	ChannelType												: UDINT := 1;(*  NC channel type:
																								1	Stantard,
																								2	Interpreter (CNC)
																								3	FIFO 
																								4	Kinematic *) 
                                        					
	EncType													: 	UDINT := E_NcEncoderType.NcEncoderType_undefined;(* Encoder type: - See property with E_NcEncoderType data type *)																																									
	EncTypAbs												:	BOOL := 0; (* Encodertyp Abs = 1/ Rel = 0*)
	
	DriveType												:	UDINT := TO_UDINT(E_NcDriveType.NcDriveType_undefined);
	
	RefFlag													:	BOOL := 0; (* Axis is in reference *)
                                							
	LimitPosActive											: 	BOOL;
	LimitNegActive											:	BOOL;
	LimitPos												: 	LREAL;
	LimitNeg												: 	LREAL;

	TargetPosWindow											:	LREAL;
	TargetPosWindowMonitoring								:	BOOL;
	PosRangeWindow											: 	LREAL;
	PosRangeWindowMonitoring								:	BOOL;
                                							
	DynamicsRefVelocity										: 	LREAL;
	DynamicsMaxVelocity										: 	LREAL;
	G0Velocity												: 	LREAL;
	RefVelocityPos											: 	LREAL;
	RefVelocityNeg											: 	LREAL;
	ManVelocityFast											: 	LREAL;
	ManVelocitySlow											: 	LREAL;
                                							  	
	Kv														: 	LREAL;
	Jerk													: 	LREAL;
	Acc														: 	LREAL;
	Dec														: 	LREAL;
	MaxPosLagValue											: 	LREAL;
	MaxPosLagFilterTime										: 	LREAL;
	MaxPosLagMonitoring										: 	BOOL;
                                                              	
	InvertEncCoutingDir										: 	BOOL;
	ModuloFactor											: 	LREAL;
	ToleranceWindowModuloStart								: 	LREAL;
	EncScalingNumerator										:	LREAL;
	EncScalingDenominator									:	LREAL;
	EncScaling												: 	LREAL; //Factor of Numerator and Denominator
	PosBias													: 	LREAL;  (* Actual NC position offset *)
	ReferenceSystem											:	UDINT; //incremental, absolute
	CalibrationMode											:	UDINT;
	CalibrationValue										: 	LREAL;	(* read/write only allowed for certain encoder types  *)
	RefFlagDistance											: 	LREAL;	(* read/write only allowed for certain encoder types *)
	CalibrInvertDirForCamSearch								:	BOOL; (* TRUE=Cam search direction negative , read/write only allowed for certain encoder types *)
	CalibrInvertDirForSyncImpSearch							:	BOOL; (* TRUE=Sync impuls (off cam) search direction negative, read/write only allowed for certain encoder types *)

	InvertMotorPolarity										: 	BOOL;
                                							  	
	BreakingDistancePos										: 	LREAL;
	BreakingDistanceNeg										: 	LREAL;
	
	PhysicalUnit											:	STRING[10+1];
END_VAR                         	


VAR
(* Zwischenspeicher ************************************************************)
	
(* Deklaration Trigger **********************************************************)

(* Zeiten ******************************************************************)

(* Bausteine ***************************************************************)
	ReadAdsPara												: ADSREAD := (NetId	:= '' , Port := AMSPORT_R0_NC, TmOut	:= DEFAULT_ADS_TIMEOUT);
	WriteAdsPara											: ADSWRITE := (NetId:= '' , Port := AMSPORT_R0_NC, TmOut	:= DEFAULT_ADS_TIMEOUT);

(* Dummy Speicher **********************************************************)

END_VAR

	(************************************************************************************)
	(*																					*)
	(*		B E C K H O F F   N E W   A U T O M A T I O N   T E C H N O L O G Y    		*)
	(*																					*)
	(*		Eiserstr.5	D-33415 Verl	Germany	phone:	+49-5246-0	www.Beckhoff.Com	*)
    (*																					*)
    (*		Bausteinbeschreibung	:	Read/Write axis parameter						*)
	(*		TwinCAT-Version			:	3.x or higher									*)
	(*																					*)
	(************************************************************************************)

(* Execute ***************************************************************************************)
	Super^();			
	
(*************************************************************************************************)

PROPERTY PROTECTED deviceAddrIsValid : BOOL
GET
deviceAddrIsValid := AxisId > 0;
END_GET
END_PROPERTY

PROPERTY PUBLIC eAxisType : E_NcAxisType
GET
eAxisType := AxisType;
END_GET
END_PROPERTY

PROPERTY PUBLIC eDriveType : E_NcDriveType
GET
eDriveType := DriveType;
END_GET
END_PROPERTY

PROPERTY PUBLIC eEncType : E_NcEncoderType
GET
eEncType := EncType;
END_GET
END_PROPERTY

METHOD PROTECTED getValue : BOOL //Return value = TRUE if execution finished and state incremented 
VAR_INPUT
	IDxGrp						:	UDINT;
	IDxOffs						:	UDINT;
	Len							:	UDINT;
	pActValue					:	PVOID; //Address of variable for actual value
	pSetValue					:	PVOID; //Address of variable for ser value variable, can be zero if no corresponding SetVariable exists
END_VAR

ReadAdsPara	(Read := TRUE, IDxGrp:=IDxGrp+AxisId, IDxOffs:=IDxOffs,LEN:=Len,DestAddr:=pActValue );
IF NOT ReadAdsPara.BUSY
THEN
	IF NOT ReadAdsPara.ERR 
	THEN 
		IF pSetValue <> 0 THEN MEMCPY(pSetValue, pActValue, Len); END_IF			
		state 												:= state + 1; 
	ELSE 		
		Busy												:= FALSE;
		Error												:= TRUE;
		ErrorId												:= ReadAdsPara.ERRID;
		ErrorText											:= CONCAT('Error read parameter in state:' , TO_STRING(state * -1));
		ErrorText											:= CONCAT(ErrorText , ' Id:');
		ErrorText											:= CONCAT(ErrorText , TO_STRING(ErrorId));
		State												:= 9999;
	END_IF	
	ReadAdsPara(Read := FALSE); 
	getValue												:= TRUE;									
END_IF
END_METHOD

METHOD PROTECTED seqRead : BOOL //Return value = TRUE if execution finished 
VAR_IN_OUT
	State							:	INT;
END_VAR
(* Execute read axis parameter ************************************)
	CASE state OF
	1..99: //read application spec parameter 
		seqRead												:= TRUE;
		
	1001: (* Name *************************************************************************************)
		IF LEN(Name) > 0 AND NOT ReadAdsPara.BUSY
		THEN
			state											:= state + 1;
		ELSE
			getValue(IDxGrp:= 16#4000,	IDxOffs := 16#2,	LEN := SIZEOF(Name),		pActValue := ADR(Name),			pSetValue := 0);
		END_IF

	1002: (* Axis Type ( Für Beschreibung Typen siehe AxPara) **********************************)
		IF AxisType <> 0 AND NOT ReadAdsPara.BUSY
		THEN
			state											:= state + 1;
		ELSE
			getValue(IDxGrp:= 16#4000,	IDxOffs := 16#3,	LEN := SIZEOF(AxisType),	pActValue := ADR(AxisType), 	pSetValue := 0);
		END_IF

	1003: (* NC Channel type ****************************************************************************************)
		IF ChannelType <> 0 AND NOT ReadAdsPara.BUSY
		THEN
			state											:= state + 1;
		ELSE
			getValue(IDxGrp:= 16#4000,	IDxOffs := 16#53,	LEN := SIZEOF(ChannelType),	pActValue := ADR(ChannelType), 	pSetValue := 0);
		END_IF

	1004: (* EncType ****************************************************************************************)
		IF EncType <> 0 AND NOT ReadAdsPara.BUSY
		THEN
			state											:= state + 1;
		ELSE
			getValue(IDxGrp:= 16#5000,	IDxOffs := 16#3,	LEN := SIZEOF(EncType),	pActValue := ADR(EncType), 		pSetValue := 0);
		END_IF
	
	1005: (* Endlagenlimit pos. ***********************************************************************)
		getValue(IDxGrp:= 16#5000,	IDxOffs := 16#E,	LEN := SIZEOF(LimitPos),	pActValue := ADR(LimitPos),  pSetValue := ADR(SetLimitPos) );	
	
	1006: (* Endlagenlimit neg ***********************************************************************)
		getValue(IDxGrp:= 16#5000,	IDxOffs := 16#D,	LEN := SIZEOF(LimitNeg),	pActValue := ADR(LimitNeg),  pSetValue := ADR(SetLimitNeg) );
		
	1007: (* Endlagenlimit pos aktiv ? ***************************************************************)
		IF getValue(IDxGrp:= 16#5000,	IDxOffs := 16#C,	LEN := SIZEOF(_UINT),	pActValue := ADR(_UINT),  pSetValue := 0)
		THEN
			SetLimitPosActive :=LimitPosActive				:= TO_BOOL(_UINT);
		END_IF

	1008: (* Endlagenlimit neg aktiv ? ***************************************************************)
		IF getValue(IDxGrp:= 16#5000,	IDxOffs := 16#B,	LEN := SIZEOF(_UINT),	pActValue := ADR(_UINT),  pSetValue := 0)
		THEN
			SetLimitNegActive :=LimitNegActive				:= TO_BOOL(_UINT);
		END_IF

	1009: (* Zielfenster ******************************************************************************)
		getValue(IDxGrp:= 16#4000,	IDxOffs := 16#16,	LEN := SIZEOF(TargetPosWindow),	pActValue := ADR(TargetPosWindow),  pSetValue := ADR(SetTargetPosWindow) );

	1010: (* Positionsfenster ************************************************************************)
		getValue(IDxGrp:= 16#4000,	IDxOffs := 16#10,	LEN := SIZEOF(PosRangeWindow),	pActValue := ADR(PosRangeWindow),  pSetValue := ADR(SetPosRangeWindow) );

	1011: (* Bezugsgeschwindigkeit (siehe Typenschild)*************************************)
		IF AxisType = 2 
		THEN
			state											:= state + 1;
		ELSE
			getValue(IDxGrp:= 16#7000,	IDxOffs := 16#101,	LEN := SIZEOF(DynamicsRefVelocity),	pActValue := ADR(DynamicsRefVelocity),  pSetValue := ADR(SetDynamicsRefVelocity) );
		END_IF
	
	1012: (* Max.Geschwindigkeit (ca. 90% der Bezugsgeschw.)***************************)
		IF AxisType = 2 
		THEN
			state											:= state + 1;
		ELSE
			getValue(IDxGrp:= 16#4000,	IDxOffs := 16#27,	LEN := SIZEOF(DynamicsMaxVelocity),	pActValue := ADR(DynamicsMaxVelocity),  pSetValue := ADR(SetDynamicsMaxVelocity) );
		END_IF
		
	1013: (* G0 Geschwindigkeit ****************************************************************)
		getValue(IDxGrp:= 16#4000,	IDxOffs := 16#A,	LEN := SIZEOF(G0Velocity),	pActValue := ADR(G0Velocity),  pSetValue := ADR(SetG0Velocity) );

	1014: (* Ref.Geschwindigkeit Pos **********************************************************)
		getValue(IDxGrp:= 16#4000,	IDxOffs := 16#6,	LEN := SIZEOF(RefVelocityPos),	pActValue := ADR(RefVelocityPos),  pSetValue := ADR(SetRefVelocityPos) );

	1015: (* Ref.Geschwindigkeit Neg **********************************************************)
		getValue(IDxGrp:= 16#4000,	IDxOffs := 16#7,	LEN := SIZEOF(RefVelocityNeg),	pActValue := ADR(RefVelocityNeg),  pSetValue := ADR(SetRefVelocityNeg) );

	1016: (* Man. Verfahrgeschwindigkeit fast *************************************************)
		getValue(IDxGrp:= 16#4000,	IDxOffs := 16#9,	LEN := SIZEOF(ManVelocityFast),	pActValue := ADR(ManVelocityFast),  pSetValue := ADR(SetManVelocityFast) );

	1017: (* Man. Verfahrgeschwindigkeit slow ***********************************************)
		getValue(IDxGrp:= 16#4000,	IDxOffs := 16#8,	LEN := SIZEOF(ManVelocitySlow),	pActValue := ADR(ManVelocitySlow),  pSetValue := ADR(SetManVelocitySlow) );

	1018: (* Kv ************************************************************************************)
		IF AxisType = 2
		THEN
			state											:= state + 1;
		ELSE
			getValue(IDxGrp:= 16#6000,	IDxOffs := 16#102,	LEN := SIZEOF(Kv),	pActValue := ADR(Kv),  pSetValue := ADR(SetKv) );
		END_IF

	1019: (* Ruck ************************************************************************************)
		IF AxisType = 2 
		THEN
			state											:= state + 1;
		ELSE
			getValue(IDxGrp:= 16#4000,	IDxOffs := 16#103,	LEN := SIZEOF(Jerk),	pActValue := ADR(Jerk),  pSetValue := ADR(SetJerk) );
		END_IF
		

	1020: (* Beschleunigung ***********************************************************************)
		IF AxisType = 2
		THEN
			state											:= state + 1;
		ELSE
			getValue(IDxGrp:= 16#4000,	IDxOffs := 16#101,	LEN := SIZEOF(Acc),	pActValue := ADR(Acc),  pSetValue := ADR(SetAcc) );
		END_IF

	1021: (* Verzoegerung ***************************************************************************)
		IF AxisType = 2 
		then
			state											:= state + 1;
		ELSE
			getValue(IDxGrp:= 16#4000,	IDxOffs := 16#102,	LEN := SIZEOF(Dec),	pActValue := ADR(Dec),  pSetValue := ADR(SetDec) );
		END_IF

	1022: (* Schleppabstand ***********************************************************************)	
		getValue(IDxGrp:= 16#6000,	IDxOffs := 16#12,	LEN := SIZEOF(MaxPosLagValue),	pActValue := ADR(MaxPosLagValue),  pSetValue := ADR(SetMaxPosLagValue) );

	1023: (* Skalierung ******************************************************************************)
		getValue(IDxGrp:= 16#5000,	IDxOffs := 16#6,	LEN := SIZEOF(EncScaling),	pActValue := ADR(EncScaling),  pSetValue := 0 );		

	1024: (* Positions Offset  ***********************************************************************)
		getValue(IDxGrp:= 16#5000,	IDxOffs := 16#7,	LEN := SIZEOF(PosBias),	pActValue := ADR(PosBias),  pSetValue := ADR(SetPosBias) );

	1025: (* Referenzposition (Nicht bei Absolut Encoder lesen)*******************************)
		IF EncType <> 2 AND EncType <> 5 AND EncType<> 7 AND EncType <> 11 AND EncType <> 12
		THEN
			getValue(IDxGrp:= 16#5000,	IDxOffs := 16#103,	LEN := SIZEOF(CalibrationValue),	pActValue := ADR(CalibrationValue),  pSetValue := ADR(SetCalibrationValue) );
		ELSE
			state											:= state +1;
		END_IF

	1026: (* Abstand Ref-Nocken Synchronimpuls (Nicht bei Absolut Encoder lesen) ****)
		IF EncType <> 2 AND EncType <> 5 AND EncType <> 7 AND EncType <> 11 AND EncType <> 12
		THEN
			getValue(IDxGrp:= 16#5100,	IDxOffs := 16#101,	LEN := SIZEOF(RefFlagDistance),	pActValue := ADR(RefFlagDistance),  pSetValue := 0 );
		ELSE
			state											:= state +1;
		END_IF

	1027: (* Drive direction **************************************************************)
		IF getValue(IDxGrp:= 16#7000,	IDxOffs := 16#6,	LEN := SIZEOF(_UINT),	pActValue := ADR(_UINT),  pSetValue := 0)
		THEN
			SetInvertMotorPolarity :=InvertMotorPolarity	:= TO_BOOL(_UINT);
			
		END_IF

	1028: (* Bremsweg positiv **********************************************************************)
		IF AxisType <> 2
		THEN
			state											:= state + 1;
		ELSE
			getValue(IDxGrp:= 16#4000,	IDxOffs := 16#303,	LEN := SIZEOF(BreakingDistancePos),	pActValue := ADR(BreakingDistancePos),  pSetValue := ADR(SetBreakingDistancePos ));
		END_IF

	1029: (* Bremsweg negativ *********************************************************************)
		IF AxisType <> 2 
		THEN
			state											:= state + 1;
		ELSE
			getValue(IDxGrp:= 16#4000,	IDxOffs := 16#304,	LEN := SIZEOF(BreakingDistanceNeg),	pActValue := ADR(BreakingDistanceNeg),  pSetValue := ADR(SetBreakingDistanceNeg ));

		END_IF

	1030: (* Schleppueberwachung Aktiv *********************************************************************)
		IF getValue(IDxGrp:= 16#6000,	IDxOffs := 16#10,	LEN := SIZEOF(_UINT),	pActValue := ADR(_UINT),  pSetValue := 0)
		THEN
			SetMaxPosLagMonitoring :=MaxPosLagMonitoring	:= TO_BOOL(_UINT);
			
		END_IF

	1031: (* Encodertyp Abs/Rel *********************************************************************)
		IF getValue(IDxGrp:= 16#5000,	IDxOffs := 16#1D,	LEN := SIZEOF(_UINT),	pActValue := ADR(_UINT),  pSetValue := 0)
		THEN
			EncTypAbs										:= TO_BOOL(_UINT);
			
		END_IF

	1032: (* Referenzierflag *********************************************************************)
		IF getValue(IDxGrp:= 16#5100,	IDxOffs := 16#9,	LEN := SIZEOF(_UINT),	pActValue := ADR(_UINT),  pSetValue := 0)
		THEN
			SetRefFlag :=RefFlag							:= TO_BOOL(_UINT);
		END_IF

	1033: (* Zielfenster Aktiv ******************************************************************)
		IF getValue(IDxGrp:= 16#4000,	IDxOffs := 16#15,	LEN := SIZEOF(_UINT),	pActValue := ADR(_UINT),  pSetValue := 0)
		THEN
			SetTargetPosWindowMonitoring :=TargetPosWindowMonitoring := TO_BOOL(_UINT);
			
		END_IF

	1034: (* Positionsfenster Aktiv ******************************************************************)
		IF getValue(IDxGrp:= 16#4000,	IDxOffs := 16#F,	LEN := SIZEOF(_UINT),	pActValue := ADR(_UINT),  pSetValue := 0)
		THEN
			SetPosRangeWindowMonitoring :=PosRangeWindowMonitoring := TO_BOOL(_UINT);
			
		END_IF

	1035: (* ModuloFaktor ******************************************************************)
		getValue(IDxGrp:= 16#5000,	IDxOffs := 16#9,	LEN := SIZEOF(ModuloFactor),	pActValue := ADR(ModuloFactor),  pSetValue := ADR(SetModuloFactor ));

	1036: (* Enc Zaehlrichtung ******************************************************************)
		IF getValue(IDxGrp:= 16#5000,	IDxOffs := 16#8,	LEN := SIZEOF(_UINT),	pActValue := ADR(_UINT),  pSetValue := 0)
		THEN
			SetInvertEncCoutingDir :=InvertEncCoutingDir := TO_BOOL(_UINT);
			
		END_IF

	1037: (* Toleranzfenster Modulo Start *******************************************************)
		getValue(IDxGrp:= 16#5000,	IDxOffs := 16#1B,	LEN := SIZEOF(ToleranceWindowModuloStart),	pActValue := ADR(ToleranceWindowModuloStart),  pSetValue := ADR(SetToleranceWindowModuloStart ));
		
	1038: (* Calibration cam search direction inverted *******************************************************)
		IF EncType <> 2 AND EncType <> 5 AND EncType<> 7 AND EncType <> 11 AND EncType <> 12
		THEN
			IF getValue(IDxGrp:= 16#5000,	IDxOffs := 16#101,	LEN := SIZEOF(_UINT),	pActValue := ADR(_UINT),  pSetValue := 0)
			THEN
				SetCalibrInvertDirForCamSearch :=CalibrInvertDirForCamSearch := TO_BOOL(_UINT);
				
			END_IF
		ELSE
			state											:= state +1;
		END_IF		
		
	1039: (* Calibration impuls direction inverted (of cam) *******************************************************)
		IF EncType <> 2 AND EncType <> 5 AND EncType<> 7 AND EncType <> 11 AND EncType <> 12
		THEN
			IF getValue(IDxGrp:= 16#5000,	IDxOffs := 16#102,	LEN := SIZEOF(_UINT),	pActValue := ADR(_UINT),  pSetValue := 0)
			THEN
				SetCalibrInvertDirForSyncImpSearch :=CalibrInvertDirForSyncImpSearch := TO_BOOL(_UINT);
				
			END_IF
	
		ELSE
			state											:= state +1;
		END_IF	
		
	1040: (* Calibration mode *******************************************************)
		IF EncType <> 2 AND EncType <> 5 AND EncType<> 7 AND EncType <> 11 AND EncType <> 12
		THEN
			getValue(IDxGrp:= 16#5000,	IDxOffs := 16#107,	LEN := SIZEOF(CalibrationMode),	pActValue := ADR(CalibrationMode),  pSetValue := ADR(SetCalibrationMode));
		ELSE
			state											:= state +1;
		END_IF
		
	1041: (* Scaling numerator **************************************)
		getValue(IDxGrp:= 16#5000,	IDxOffs := 16#23,	LEN := SIZEOF(EncScalingNumerator),	pActValue := ADR(EncScalingNumerator),  pSetValue := ADR(SetEncScalingNumerator) );	
			
	1042: (* Scaling denumerator **************************************)
		getValue(IDxGrp:= 16#5000,	IDxOffs := 16#24,	LEN := SIZEOF(EncScalingDenominator),	pActValue := ADR(EncScalingDenominator),  pSetValue := ADR(SetEncScalingDenominator) );	
		
	1043: (* Reference system **************************************)
		getValue(IDxGrp:= 16#5000,	IDxOffs := 16#19,	LEN := SIZEOF(ReferenceSystem),	pActValue := ADR(ReferenceSystem),  pSetValue := ADR(SetReferenceSystem) );	

	1044: (* Schleppabstand Filter Time ***********************************************************************)	
		getValue(IDxGrp:= 16#6000,	IDxOffs := 16#13,	LEN := SIZEOF(MaxPosLagFilterTime),	pActValue := ADR(MaxPosLagFilterTime),  pSetValue := ADR(SetMaxPosLagFilterTime) );

	1045: (* Physical unit ***********************************************************************)	
		getValue(IDxGrp:= 16#4000,	IDxOffs := 16#5,	LEN := SIZEOF(PhysicalUnit),	pActValue := ADR(PhysicalUnit),  pSetValue := ADR(PhysicalUnit) );
		IF PhysicalUnit[0] = 176 THEN PhysicalUnit := '°'; END_IF		
		
	1046: (*  Drive type ***********************************************************************)	
		getValue(IDxGrp:= 16#7000,	IDxOffs := 16#3,	LEN := SIZEOF(DriveType),	pActValue := ADR(DriveType),  pSetValue := 0 );
			
	ELSE
		state												:= 1;
	END_CASE

(*********************************************************************************************)
END_METHOD

METHOD PROTECTED seqWrite : BOOL //Return value = TRUE if execution finished 
VAR_IN_OUT
	State							:	INT;
END_VAR
(* Write axis parameter ********************************************************************)
	CASE state OF
	1..99: //Wite application spec parameter 
		seqWrite											:= TRUE;
		
	1001: (* Endlagenlimit pos.beschreiben ********************************************************)
		setValue(IDxGrp:= 16#5000,	IDxOffs := 16#E,	LEN := SIZEOF(SetLimitPos),		pActValue := ADR(LimitPos),		pSetValue := ADR(SetLimitPos));

	1002: (* Endlagenlimit neg.beschreiben ********************************************************)
		setValue(IDxGrp:= 16#5000,	IDxOffs := 16#D,	LEN := SIZEOF(SetLimitNeg),		pActValue := ADR(LimitNeg),		pSetValue := ADR(SetLimitNeg));

	1003: (* Endlagenlimit pos. aktiv ****************************************************************)
		IF NOT (SetLimitPosActive XOR LimitPosActive)
			AND NOT WriteAdsPara.BUSY
		THEN 
			state 											:= state + 1;
		ELSE
			_UINT											:= TO_UINT(SetLimitPosActive);
			LimitPosActive									:= SetLimitPosActive;
			setValue(IDxGrp:= 16#5000,	IDxOffs := 16#C,	LEN := SIZEOF(_UINT),		pActValue := 0,		pSetValue := ADR(_UINT));
		END_IF
		
	1004: (* Endlagenlimit neg.aktiv *****************************************************************)
		IF NOT (SetLimitNegActive XOR LimitNegActive) 
			AND NOT WriteAdsPara.BUSY
		THEN 
			state 											:= state + 1;
		ELSE
			_UINT											:= TO_UINT(SetLimitNegActive);
			LimitNegActive									:= SetLimitNegActive; 
			setValue(IDxGrp:= 16#5000,	IDxOffs := 16#B,	LEN := SIZEOF(_UINT),		pActValue := 0,		pSetValue := ADR(_UINT));
		END_IF

	1005: (* Zielfenster setzen **********************************************************************)
		setValue(IDxGrp:= 16#4000,	IDxOffs := 16#16,	LEN := SIZEOF(SetTargetPosWindow),		pActValue := ADR(TargetPosWindow),		pSetValue := ADR(SetTargetPosWindow));

	1006: (* Positionsfenster setzen *****************************************************************)
		setValue(IDxGrp:= 16#4000,	IDxOffs := 16#10,	LEN := SIZEOF(SetPosRangeWindow),		pActValue := ADR(PosRangeWindow),	pSetValue := ADR(SetPosRangeWindow));
		
	1007: (* Bezugsgeschwindigkeit setzen ********************************************************)
		IF AxisType = 2
		THEN 
			state 											:= state +1;
		ELSE
			setValue(IDxGrp:= 16#7000,	IDxOffs := 16#101,	LEN := SIZEOF(SetDynamicsRefVelocity),pActValue := ADR(DynamicsRefVelocity),	pSetValue := ADR(SetDynamicsRefVelocity));
		END_IF


	1008: (* Max.Geschwindigkeit setzen ************************************************************)
		IF AxisType = 2 
		THEN 
			state 											:= state +1;
		ELSE
			setValue(IDxGrp:= 16#4000,	IDxOffs := 16#27,	LEN := SIZEOF(SetDynamicsMaxVelocity),pActValue := ADR(DynamicsMaxVelocity),	pSetValue := ADR(SetDynamicsMaxVelocity));
		END_IF

	1009: (* G0 Geschwindigkeit setzen ****************************************************************)
		setValue(IDxGrp:= 16#4000,	IDxOffs := 16#A,	LEN := SIZEOF(SetG0Velocity),	pActValue := ADR(G0Velocity),	pSetValue := ADR(SetG0Velocity));

	1010: (* Ref.Geschwindigkeit fast setzen *******************************************************)
		setValue(IDxGrp:= 16#4000,	IDxOffs := 16#6,	LEN := SIZEOF(SetRefVelocityPos),	pActValue := ADR(RefVelocityPos),	pSetValue := ADR(SetRefVelocityPos));

	1011: (* Ref.Geschwindigkeit slow setzen *****************************************************)
		setValue(IDxGrp:= 16#4000,	IDxOffs := 16#7,	LEN := SIZEOF(SetRefVelocityNeg),	pActValue := ADR(RefVelocityNeg),	pSetValue := ADR(SetRefVelocityNeg));

	1012: (* Man.Geschwindigkeit fast setzen ******************************************************)
		setValue(IDxGrp:= 16#4000,	IDxOffs := 16#9,	LEN := SIZEOF(SetManVelocityFast),	pActValue := ADR(ManVelocityFast),	pSetValue := ADR(SetManVelocityFast));
		

	1013: (* Man.Geschwindigkeit slow setzen ******************************************************)
		setValue(IDxGrp:= 16#4000,	IDxOffs := 16#8,	LEN := SIZEOF(SetManVelocitySlow),	pActValue := ADR(ManVelocitySlow),	pSetValue := ADR(SetManVelocitySlow));

	1014: (* Kv setzen **************************************************************************************)
		IF AxisType = 2 
		THEN 
			state 											:= state +1;
		ELSE
			setValue(IDxGrp:= 16#6000,	IDxOffs := 16#102,	LEN := SIZEOF(SetKv),pActValue := ADR(Kv),	pSetValue := ADR(SetKv));
		END_IF

	1015: (* Ruck setzen ***********************************************************************************)
		IF AxisType = 2 
		THEN 
			state 											:= state +1;
		ELSE
			setValue(IDxGrp:= 16#4000,	IDxOffs := 16#103,	LEN := SIZEOF(SetJerk),pActValue := ADR(Jerk),	pSetValue := ADR(SetJerk));
		END_IF

	1016: (* Beschleunigung setzen **********************************************************************)
		IF AxisType = 2 
		THEN 
			state 											:= state +1;
		ELSE
			setValue(IDxGrp:= 16#4000,	IDxOffs := 16#101,	LEN := SIZEOF(SetAcc), pActValue := ADR(Acc),	pSetValue := ADR(SetAcc));
		END_IF
	
	1017: (* Verzoegerung setzen ************************************************************************)
		IF AxisType = 2 
		THEN 
			state 											:= state +1;
		ELSE
			setValue(IDxGrp:= 16#4000,	IDxOffs := 16#102,	LEN := SIZEOF(SetDec), pActValue := ADR(Dec),	pSetValue := ADR(SetDec));
		END_IF
		
	1018: (* Schleppabstand setzen **********************************************************************)
		setValue(IDxGrp:= 16#6000,	IDxOffs := 16#12,	LEN := SIZEOF(SetMaxPosLagValue),	pActValue := ADR(MaxPosLagValue),	pSetValue := ADR(SetMaxPosLagValue));

	1019: (* Reserverd *****************************************************************************)
		// Set scaling replaced by Num and Denum  setValue(IDxGrp:= 16#5000,	IDxOffs := 16#6,	LEN := SIZEOF(SetEncScaling),	pActValue := ADR(EncScaling),	pSetValue := ADR(SetEncScaling));
		state 												:= state +1 ;
		
	1020: (* Positions Offset setzen ****************************************************************)
		setValue(IDxGrp:= 16#5000,	IDxOffs := 16#7,	LEN := SIZEOF(SetPosBias),	pActValue := ADR(PosBias),	pSetValue := ADR(SetPosBias));
		
	1021: (* Referenzposition setzen ***************************************************************)
		IF EncType <> 2  AND EncType <> 5 AND EncType <> 7 AND EncType <> 11  AND EncType <> 12 
		THEN
			setValue(IDxGrp:= 16#5000,	IDxOffs := 16#103,	LEN := SIZEOF(SetCalibrationValue),	pActValue := ADR(CalibrationValue),	pSetValue := ADR(SetCalibrationValue));
		ELSE
			state 											:= state +1 ;
		END_IF

	1022: (* Bremsweg positiv **********************************************************************)
		IF AxisType = 2 
		THEN 
			state 											:= state +1;
		ELSE
			setValue(IDxGrp:= 16#4000,	IDxOffs := 16#303,	LEN := SIZEOF(SetBreakingDistancePos), pActValue := ADR(BreakingDistancePos),	pSetValue := ADR(SetBreakingDistancePos));
		END_IF

	1023: (* Bremsweg negativ *********************************************************************)
		IF AxisType = 2
		THEN 
			state 											:= state +1;
		ELSE
			setValue(IDxGrp:= 16#4000,	IDxOffs := 16#304,	LEN := SIZEOF(SetBreakingDistanceNeg), pActValue := ADR(BreakingDistanceNeg),	pSetValue := ADR(SetBreakingDistanceNeg));
		END_IF

	1024: (* Schleppueberwachung ****************************************************************************)
		IF SetMaxPosLagMonitoring = MaxPosLagMonitoring AND NOT WriteAdsPara.BUSY
		THEN 
			state 											:= state +1;
		ELSE
			_UINT											:= TO_UINT(SetMaxPosLagMonitoring);
			MaxPosLagMonitoring								:= SetMaxPosLagMonitoring;					
			setValue(IDxGrp:= 16#6000,	IDxOffs := 16#10,	LEN := SIZEOF(_UINT),	pActValue := 0,	pSetValue := ADR(_UINT));
		END_IF

	1025: (* Referenzierflag ****************************************************************************)
		IF RefFlag = SetRefFlag AND NOT WriteAdsPara.BUSY
		THEN 
			state 											:= state +1;
		ELSE
			_UINT											:= TO_UINT(SetRefFlag);
			RefFlag											:= SetRefFlag;
			setValue(IDxGrp:= 16#5100,	IDxOffs := 16#9,	LEN := SIZEOF(_UINT), pActValue := 0,	pSetValue := ADR(_UINT));
		END_IF
		
	1026: (* PosfensterAktiv ****************************************************************************)
		IF SetPosRangeWindowMonitoring = PosRangeWindowMonitoring AND NOT WriteAdsPara.BUSY
		THEN 
			state 											:= state +1;
		ELSE
			_UINT											:= TO_UINT(SetPosRangeWindowMonitoring);
			PosRangeWindowMonitoring						:= SetPosRangeWindowMonitoring;
			setValue(IDxGrp:= 16#4000,	IDxOffs := 16#F,	LEN := SIZEOF(_UINT), pActValue := 0,	pSetValue := ADR(_UINT));
		END_IF

	1027: (* ZielfensterAktiv ****************************************************************************)
		IF SetTargetPosWindowMonitoring = TargetPosWindowMonitoring AND NOT WriteAdsPara.BUSY
		THEN 
			state 											:= state +1;
		ELSE
			_UINT											:= TO_UINT(SetTargetPosWindowMonitoring);
			TargetPosWindowMonitoring						:= SetTargetPosWindowMonitoring;
			setValue(IDxGrp:= 16#4000,	IDxOffs := 16#15,	LEN := SIZEOF(_UINT), pActValue := 0,	pSetValue := ADR(_UINT));
		END_IF

	1028: (* Modulofaktor ****************************************************************************)
		setValue(IDxGrp:= 16#5000,	IDxOffs := 16#9,	LEN := SIZEOF(SetModuloFactor), pActValue := ADR(ModuloFactor),	pSetValue := ADR(SetModuloFactor));
		
	1029: (* Enc. Zaehlrichtung ****************************************************************************)
		IF SetInvertEncCoutingDir = InvertEncCoutingDir AND NOT WriteAdsPara.BUSY
		THEN 
			state 											:= state +1;
		ELSE
			_UINT											:= TO_UINT(SetInvertEncCoutingDir);
			InvertEncCoutingDir								:= SetInvertEncCoutingDir;
			setValue(IDxGrp:= 16#5000,	IDxOffs := 16#8,	LEN := SIZEOF(_UINT), pActValue := 0,	pSetValue := ADR(_UINT));
		END_IF

	1030: (* Drive  ****************************************************************************)
		IF SetInvertMotorPolarity = InvertMotorPolarity AND NOT WriteAdsPara.BUSY
		THEN 
			state 											:= state +1;
		ELSE
			_UINT											:= TO_UINT(SetInvertMotorPolarity);
			InvertMotorPolarity								:= SetInvertMotorPolarity;
			setValue(IDxGrp:= 16#7000,	IDxOffs := 16#6,	LEN := SIZEOF(_UINT), pActValue := 0,	pSetValue := ADR(_UINT));
		END_IF
		
		
	1031: (* Enc. Modulo start tolerance ****************************************************************************)
		setValue(IDxGrp:= 16#5000,	IDxOffs := 16#1B,	LEN := SIZEOF(SetToleranceWindowModuloStart), pActValue := ADR(ToleranceWindowModuloStart),	pSetValue := ADR(SetToleranceWindowModuloStart));

	1032: (* Set calibration cam search direction inverted ***************************************************************)
		IF SetCalibrInvertDirForCamSearch = CalibrInvertDirForCamSearch	AND NOT WriteAdsPara.BUSY
			OR_ELSE(EncType = 2  OR EncType = 5 OR EncType = 7 OR EncType = 11  OR EncType = 12)
		THEN 
			state 											:= state +1;
		ELSE
			_UINT											:= TO_UINT(SetCalibrInvertDirForCamSearch);
			CalibrInvertDirForCamSearch						:= SetCalibrInvertDirForCamSearch;
			setValue(IDxGrp:= 16#5000,	IDxOffs := 16#101,	LEN := SIZEOF(_UINT), pActValue := 0,	pSetValue := ADR(_UINT));
		END_IF

	1033: (* Set calibration impuls search direction inverted ***************************************************************)
		IF SetCalibrInvertDirForSyncImpSearch = CalibrInvertDirForSyncImpSearch AND NOT WriteAdsPara.BUSY
			OR_ELSE(EncType = 2  OR EncType = 5 OR EncType = 7 OR EncType = 11  OR EncType = 12)
		THEN 
			state 											:= state +1;
		ELSE
			_UINT											:= TO_UINT(SetCalibrInvertDirForSyncImpSearch);
			CalibrInvertDirForSyncImpSearch					:= SetCalibrInvertDirForSyncImpSearch;
			setValue(IDxGrp:= 16#5000,	IDxOffs := 16#102,	LEN := SIZEOF(_UINT), pActValue := 0,	pSetValue := ADR(_UINT));
		END_IF
		
	1034: (* Set calibration mode ***************************************************************)
		IF SetCalibrationMode = CalibrationMode  AND NOT WriteAdsPara.BUSY
			OR_ELSE(EncType = 2  OR EncType = 5 OR EncType = 7 OR EncType = 11  OR EncType = 12)
		THEN 
			state 											:= state +1;		
		ELSE
			setValue(IDxGrp:= 16#5000,	IDxOffs := 16#107,	LEN := SIZEOF(SetCalibrationMode), pActValue := ADR(CalibrationMode),	pSetValue := ADR(SetCalibrationMode));
		END_IF

	1035: (* Scaling numerator **************************************)
		setValue(IDxGrp:= 16#5000,	IDxOffs := 16#23,	LEN := SIZEOF(SetEncScalingNumerator),	pActValue := ADR(EncScalingNumerator),  pSetValue := ADR(SetEncScalingNumerator) );	
			
	1036: (* Scaling denumerator **************************************)
		setValue(IDxGrp:= 16#5000,	IDxOffs := 16#24,	LEN := SIZEOF(SetEncScalingDenominator),	pActValue := ADR(EncScalingDenominator),  pSetValue := ADR(SetEncScalingDenominator) );
		
		//Calculate Act Scaling 
		IF NOT Error THEN  EncScaling	:= EncScalingNumerator / EncScalingDenominator; END_IF
		
	1037: (* Reference system **************************************)
		setValue(IDxGrp:= 16#5000,	IDxOffs := 16#19,	LEN := SIZEOF(SetReferenceSystem),	pActValue := ADR(ReferenceSystem),  pSetValue := ADR(SetReferenceSystem) );	
	
	1038: (* Schleppueberwachung Zeit ****************************************************************************)
		setValue(IDxGrp:= 16#6000,	IDxOffs := 16#13,	LEN := SIZEOF(SetMaxPosLagFilterTime),	pActValue := ADR(MaxPosLagFilterTime),	pSetValue := ADR(SetMaxPosLagFilterTime));
	
	ELSE
		state 												:= 1 ;
	END_CASE
	
(***********************************************************************************************)
END_METHOD

METHOD PROTECTED setValue : BOOL //Return value = TRUE if execution finished and state incremented 
VAR_INPUT
	IDxGrp						:	UDINT;
	IDxOffs						:	UDINT;
	Len							:	UDINT;
	pActValue					:	PVOID; //Address of variable for actual value, can be zero if no corresponding acual value variable exists
	pSetValue					:	PVOID; //Address of variable for set value variable
END_VAR

IF pActValue <> 0 AND pSetValue <> 0 AND_THEN MEMCMP(pSetValue, pActValue, Len) = 0
THEN //Skip write parameter if set and actual value are equel
	state													:= state + 1;	
	setValue												:= TRUE;
ELSE
	WriteAdsPara( Write := TRUE, IdxGrp :=IDxGrp+AxisId, IdxOffs:=IDxOffs, LEN:=Len, SrcAddr:=pSetValue );
	IF NOT WriteAdsPara.BUSY
	THEN
		IF NOT WriteAdsPara.ERR
		THEN
			IF pActValue <> 0 THEN MEMCPY(pActValue, pSetValue, Len); END_IF	
			state											:= state + 1;
		ELSE
			Busy											:= FALSE;
			Error											:= TRUE;
			ErrorId											:= WriteAdsPara.ERRID;
			ErrorText										:= CONCAT('Error write parameter in state:' , TO_STRING(state * -1));
			ErrorText										:= CONCAT(ErrorText , ' Id:');
			ErrorText										:= CONCAT(ErrorText , TO_STRING(ErrorId));
			State											:= 9999;
		END_IF
		WriteAdsPara (Write := FALSE);
		setValue											:= TRUE;
	END_IF		
END_IF
END_METHOD

END_FUNCTION_BLOCK

// ---- POUs/Motion/TF5100-NCI/NciChannel_wEvents.TcPOU
{attribute 'no_check'}
FUNCTION_BLOCK NciChannel_wEvents EXTENDS NciChannel
VAR_INPUT

                        								      
	Event													:	NciEventHandling;
                        	
END_VAR                 	
VAR_OUTPUT              	

END_VAR
VAR
END_VAR

	(* NCI Control											*)
	(********************************************************)

(********************************************************************************)
(* error event ctrl																*)
(********************************************************************************)
	Event(
		Enable			:= ,
		ConfirmTrig		:= NOT Errhdl.flag AND Event.Status.31 OR Admin.ResetAdmin,
		Name			:= ErrHdl.fnc,
		SourceId		:= (* Default *) ,
		rNci			:= THIS^,
		ErrorId			:= TO_UDINT(ErrHdl.Id),
		Status			=> );
		
	(* Reset FB errors by reset flag *)
	(* currently not in use, call _Resetting via state machine to reset Fb errors by setting Execute to FALSE 
	IF Admin.Reset
	THEN
		grp.Execute											:= grp.Execute AND NOT grp.Error;
		itp.Execute											:= itp.Execute AND NOT itp.Error;
		Motion.Execute										:= Motion.Execute AND NOT Motion.Error;
		RPara.Execute										:= RPara.Execute AND NOT RPara.Error;
	END_IF
	*)
	
(********************************************************************************)
(* call super 																	*)
(********************************************************************************)
	SUPER^();
(******************************************************************************)

METHOD reset : Bool
VAR_INPUT
END_VAR

reset 			:= ErrHdl.flag OR SUPER^.reset();
Event.confirm();
END_METHOD

END_FUNCTION_BLOCK

// ---- POUs/Motion/TF5100-NCI/NciChannel.TcPOU
{attribute 'no_check'}
FUNCTION_BLOCK NciChannel EXTENDS NCI_REF
VAR_INPUT
	Admin													:	NciAdmin;
	grp														:	NciGrp;
	Itp														:	NciItp;
	motion													:	NciMotion;
                        								   
	MFnc													: 	NciMFnc;
	RPara													:	NciReadWriteRParam;
                        	
END_VAR                 	
VAR_OUTPUT              	
	ErrHdl													:	ERROR_HDL;
END_VAR
VAR
END_VAR

	(* NCI Control											*)
	(********************************************************)

(********************************************************************************)
(* work admin ctrl																*)
(********************************************************************************)
	admin(
		ResetAdmin				:= ,
		Enable					:= ,
		EStop					:= ,
		SingleBlockMode			:= , 
		InSingleBlockTrigNext	:= , 
		GrpCnfg					:= ,
		Override				:= ,
		SpindleOvr				:= ,	
		rNCIRef					:= THIS^,
		InGroup					=> ,
		Busy					=> ,
		Done					=> ,
		Error					=> ,
		ErrorID					=> ,
		ErrorText				=> );

(********************************************************************************)
(* work group ctrl																*)
(********************************************************************************)
	grp(
		Execute				:= ,
		Fnc					:= ,
		XAxisId				:= ,
		YAxisId				:= ,
		ZAxisId				:= ,
		Q1AxisId			:= ,
		Q2AxisId			:= ,
		Q3AxisId			:= ,
		Q4AxisId			:= ,
		Q5AxisId			:= ,
		AxisIndex			:= ,
		rNCIRef				:= THIS^, 
		Busy				=> ,
		Done				=> ,
		Error				=> ,
		ErrorID				=> ,
		ErrorText			=> );

(********************************************************************************)
(* work interpolation ctrl														*)
(********************************************************************************)
	Itp(
		Execute				:= ,
		Fnc					:= ,
		Prg					:= ,
		rTable				:= ,
		rNCIRef				:= THIS^,
		StartPrgAfterLoading:= , 
		LogFeederEntries	:= ,
		Busy				=> ,
		Done				=> ,
		Error				=> ,
		ErrorID				=> ,
		ErrorText			=> );


(********************************************************************************)
(* work motion ctrl																*)
(********************************************************************************)
	motion(
		Execute						:= ,
		Fnc							:= ,
		rNCIRef						:= THIS^,
		FNC_ESTOP					=> ,
		FNC_STEP_ON					=> ,
		FNC_ENABLE_FEEDER_BACKUP	=> ,
		FNC_DISABLE_FEEDER_BACKUP	=> ,
		FNC_RETRACE_FWD				=> ,
		FNC_RETRACE_BWD				=> ,
		Busy						=> ,
		Done						=> ,
		Error						=> ,
		ErrorId						=> ,
		ErrorText					=> );

(********************************************************************************)
(* work R rarameter ctrl														*)
(********************************************************************************)
	RPara(
		Execute						:= ,
		Fnc							:= ,
		pAddr						:= ,
		Index						:= ,
		Count						:= ,
		rNCIRef						:= THIS^,
		Done						=> ,
		Busy						=> ,
		Error						=> ,
		ErrorId						=> );

(********************************************************************************)
(* work M function  ctrl														*)
(********************************************************************************)
	MFnc(
		ConfirmHsk					:= ,
		FastMFuncReset				:= ,
		FastMFuncNo					:= ,
		rNCIRef						:= THIS^);

(********************************************************************************)
(* collect errors																*)
(********************************************************************************)
	IF Admin.Error
	THEN
		ErrHdl.flag											:= Admin.Error;
		ErrHdl.id											:= UDINT_TO_DINT(Admin.ErrorID);
		ErrHdl.fnc											:= 'NciAdmin';
		ErrHdl.text											:= Admin.ErrorText;
                        									
	ELSIF grp.Error     									
	THEN                									
		ErrHdl.flag											:= grp.Error;
		ErrHdl.id											:= UDINT_TO_DINT(grp.ErrorID);
		ErrHdl.fnc											:= 'NciGrp';
		ErrHdl.text											:= grp.ErrorText;
                        									
	ELSIF itp.Error     									
	THEN                									
		ErrHdl.flag											:= Itp.Error;
		ErrHdl.id											:= UDINT_TO_DINT(Itp.ErrorID);
		ErrHdl.fnc											:= 'NciItp';
		ErrHdl.text											:= Itp.ErrorText;
                        									
	ELSIF motion.Error  									
	THEN                									
		ErrHdl.flag											:= motion.Error;
		ErrHdl.id											:= UDINT_TO_DINT(motion.ErrorID);
		ErrHdl.fnc											:= 'NciMotion';
		ErrHdl.text											:= motion.ErrorText;
		
	ELSIF RPara.Error  									
	THEN                									
		ErrHdl.flag											:= RPara.Error;
		ErrHdl.id											:= UDINT_TO_DINT(RPara.ErrorID);
		ErrHdl.fnc											:= 'RPara';
		ErrHdl.text											:= CONCAT('Error RPara id: ',  UDINT_TO_STRING(RPara.Errorid));
	ELSE
		ErrHdl.Reset();
	END_IF
(******************************************************************************)

METHOD PUBLIC noAction : BOOL
VAR_INPUT
END_VAR
grp.Execute													:= FALSE;
itp.Execute													:= FALSE;
Motion.Execute												:= FALSE;
RPara.Execute												:= FALSE;

NoAction 													:= NOT Grp.Busy and not Itp.Busy and not Motion.Busy and not RPara.Busy;
END_METHOD

METHOD reset : Bool
VAR_INPUT
END_VAR
NoAction();
reset 			:= Admin.reset(FALSE);
END_METHOD

END_FUNCTION_BLOCK

// ---- POUs/Motion/TF5100-NCI/01_Main/NciAdmin.TcPOU
{attribute 'no_check'}
//NCI group administration - Build/Reconfig group via Enable input, activate EStop and StepOn after releasing EStop input
//based on Tc2_NCI library
FUNCTION_BLOCK NciAdmin
VAR_INPUT
	ResetAdmin												:	BOOL := FALSE; (* Reset Nci group *)
	Enable													:	BOOL := FALSE; (* TRUE = Build Group / FALSE = Reconfig Group *)
	EStop													:	BOOL := FALSE; (* TRUE = EStop / FALSE = StepOn *)
	SingleBlockMode											:	E_ItpSingleBlockMode := ItpSingleBlockOff; (* Operation mode for single set:
																											 	ItpSingleBlockOff: single set off
																											 	ItpSingleBlockNck: single set in the NC kernel 
																												ItpSingleBlockIntp: single set in the interpreter *)
	InSingleBlockTrigNext									:	BOOL	:= FALSE;
	GrpCnfg													:	NCI_EXT3DGROUP;
	Override												:	LREAL := 0.0; //0.0-100.0%
	SpindleOvr												:	LREAL := 0.0; //0.0-100.0%
	rNCIRef													:	REFERENCE TO NCI_REF := 0;
END_VAR
VAR_IN_OUT
END_VAR
VAR_OUTPUT
	InGroup													:	BOOL; 
	Busy													:	BOOL;
	Done													:	BOOL;
	Error													:	BOOL;
{attribute 'displaymode':='hex'}
	ErrorID													:	UDINT;
	ErrorText												:	STRING(40);
END_VAR
VAR
(* Zwischenspeicher **************************************************************************)
	MemDone													:	BOOL;
	MemFnc													:	INT := 0;

(* Instanzierung der MC Bausteine *******************************************************)
	ItpSingleBlock											:	ItpSingleBlock := (tTimeOut	:= DEFAULT_ADS_TIMEOUT);
	CfgBuildExt3DGroup										:	CfgBuildExt3DGroup := (tTimeOut	:= DEFAULT_ADS_TIMEOUT);
	CfgReconfigGroup										:	CfgReconfigGroup := (tTimeOut	:= DEFAULT_ADS_TIMEOUT);
	ItpResetEx2												:	ItpResetEx2 := (tTimeOut	:= DEFAULT_ADS_TIMEOUT);
	ItpEStopEx												:	ItpEStopEx := (tTimeOut	:= DEFAULT_ADS_TIMEOUT);
	ItpStepOnAfterEStopEx									:	ItpStepOnAfterEStopEx := (tTimeOut	:= DEFAULT_ADS_TIMEOUT);

(* Dummy  **********************************************************)
	Dummy 	: BOOL;
END_VAR

	(* NCI group administration															*)
	(************************************************************************************)

(* verify reference ***********************************************************************)
IF NOT __ISVALIDREF(rNCIRef) 
THEN
	Busy													:= NOT Error;
	ErrorId													:= E_AdsErr.DEVICE_INVALIDPARM;
	Error													:= TRUE;
	Done													:= FALSE;
	InGroup													:= FALSE;
	ErrorText												:= 'Reference to rNCIRef invalid (0)';
	RETURN;
END_IF

(* reading axis-status from NCtoPLC-channel *************************************************)
	rNCIRef.ReadStatus();

(* writing override into the NC-interface ***************************************************)
	rNCIRef.PlcToNci.ChnAxesOvr 							:= LREAL_TO_DWORD(LIMIT(0.0,Override,100.0) * 10000.0 );
	rNCIRef.PlcToNci.ChnSpindleOvr							:= LREAL_TO_DWORD(LIMIT(0.0,SpindleOvr,100.0) * 10000.0 );

(* Build Grp / rebuild grp ******************************************************************)
	InGroup													:=  NOT CfgBuildExt3DGroup.bBusy 
																AND(rNCIRef.NciToPlc.AcsAxisIDs[0] = GrpCnfg.nXAxisId 		
																AND rNCIRef.NciToPlc.AcsAxisIDs[1] = GrpCnfg.nYAxisId 
																and rNCIRef.NciToPlc.AcsAxisIDs[2] = GrpCnfg.nZAxisId 
																and rNCIRef.NciToPlc.AcsAxisIDs[3] = GrpCnfg.nQ1AxisId
																and rNCIRef.NciToPlc.AcsAxisIDs[4] = GrpCnfg.nQ2AxisId
																and rNCIRef.NciToPlc.AcsAxisIDs[5] = GrpCnfg.nQ3AxisId
																and rNCIRef.NciToPlc.AcsAxisIDs[6] = GrpCnfg.nQ4AxisId
																AND rNCIRef.NciToPlc.AcsAxisIDs[7] = GrpCnfg.nQ5AxisId																
																OR  
																rNCIRef.NciToPlc.McsAxisIDs[0] = GrpCnfg.nXAxisId 
																AND rNCIRef.NciToPlc.McsAxisIDs[1] = GrpCnfg.nYAxisId 
																and rNCIRef.NciToPlc.McsAxisIDs[2] = GrpCnfg.nZAxisId 
																and rNCIRef.NciToPlc.McsAxisIDs[3] = GrpCnfg.nQ1AxisId
																and rNCIRef.NciToPlc.McsAxisIDs[4] = GrpCnfg.nQ2AxisId
																and rNCIRef.NciToPlc.McsAxisIDs[5] = GrpCnfg.nQ3AxisId
																and rNCIRef.NciToPlc.McsAxisIDs[6] = GrpCnfg.nQ4AxisId
																AND rNCIRef.NciToPlc.McsAxisIDs[7] = GrpCnfg.nQ5AxisId);
							
	Dummy													:= CfgBuildExt3DGroup.bBusy; //Catch busy status before next call of FB
									
	CfgBuildExt3DGroup(
		bExecute	:= Enable AND NOT CfgReconfigGroup.bBusy,
		nGroupId	:= rNCIRef.NciToPlc.GrpId,
		nXAxisId	:= GrpCnfg.nXAxisId,
		nYAxisId	:= GrpCnfg.nYAxisId,
		nZAxisId	:= GrpCnfg.nZAxisId,
		nQ1AxisId	:= GrpCnfg.nQ1AxisId,
		nQ2AxisId	:= GrpCnfg.nQ2AxisId,
		nQ3AxisId	:= GrpCnfg.nQ3AxisId,
		nQ4AxisId	:= GrpCnfg.nQ4AxisId,
		nQ5AxisId	:= GrpCnfg.nQ5AxisId,
		tTimeOut	:= ,
		bBusy		=> ,
		bErr		=> ,
		nErrId		=> );

	IF 	Dummy 
		AND NOT CfgBuildExt3DGroup.bBusy 
		AND NOT CfgBuildExt3DGroup.bErr
	THEN
	//	InGroup												:= TRUE;
		MemDone												:= TRUE;
	END_IF


	(* Reconfig Grp *)
	Dummy													:= CfgReconfigGroup.bBusy;

	CfgReconfigGroup(
		bExecute	:= NOT Enable AND NOT CfgBuildExt3DGroup.bBusy AND(InGroup OR CfgReconfigGroup.bErr AND NOT Memfnc.7 ),
		nGroupId	:= rNCIRef.NciToPlc.GrpId,
		tTimeOut	:= ,
		bBusy		=> ,
		bErr		=> ,
		nErrId		=> );

	IF 	Dummy 
		AND NOT CfgReconfigGroup.bBusy 
		AND NOT CfgReconfigGroup.bErr
	THEN
	//	InGroup												:= FALSE;
		MemDone												:= TRUE;
	END_IF


(* Estop ****************************************************************************************)
	Dummy													:= ItpEStopEx.bBusy;

	ItpEStopEx(
		bExecute	:= EStop AND NOT ItpStepOnAfterEStopEx.bBusy,
		fDec		:= (* Dec *),
		fJerk		:= (* Jerk *),
		tTimeOut	:= ,
		sNciToPlc	:= rNCIRef.NciToPlc,
		bBusy		=> ,
		bErr		=> ,
		nErrId		=> );
		
	IF ItpEStopEx.bExecute
	THEN //Triggerd by input
		MemFnc.0											:= TRUE;
	END_IF

	IF 	Dummy 
		AND NOT ItpEStopEx.bBusy 
	THEN
		MemDone												:= NOT ItpEStopEx.bErr;
	END_IF

	(* Step on after estop *)
	Dummy													:= ItpStepOnAfterEStopEx.bBusy;
	
	ItpStepOnAfterEStopEx(
		bExecute	:= NOT ItpEStopEx.bExecute AND NOT ItpEStopEx.bBusy AND rNCIRef.NciToPlc.ChnState.8 AND memFnc.0, //EStopReq ,
		tTimeOut	:= ,
		sNciToPlc	:= rNCIRef.NciToPlc,
		bBusy		=> ,
		bErr		=> ,
		nErrId		=> );

	IF 	Dummy 
		AND NOT ItpStepOnAfterEStopEx.bBusy 
	THEN
		MemDone												:= NOT ItpStepOnAfterEStopEx.bErr;
		MemFnc.0											:= FALSE;
	END_IF
	
(* Method fnc ****************************************************************)
	IF NOT Memfnc.4 
	THEN
		IF ResetAdmin
		THEN			
			MemFnc.4										:= reset(Execute:= TRUE);
		END_IF
	ELSIF NOT reset(Execute:= ResetAdmin)
	THEN
		MemDone												:= TRUE;
		MemFnc.4											:= FALSE;
	END_IF
	
	IF NOT Memfnc.5
	THEN
		IF SingleBlockMode <> ItpSingleBlock.nMode 
		THEN
			MemFnc.5										:= SingleBlockModeChange(Execute:= TRUE,SingleBlockMode := SingleBlockMode);
		END_IF
	ELSIF NOT SingleBlockModeChange(Execute:= FALSE, SingleBlockMode := SingleBlockMode)
	THEN
		MemDone												:= TRUE;
		MemFnc.5											:= FALSE;
	END_IF

	IF NOT Memfnc.6
	THEN
		IF InSingleBlockTrigNext
		THEN
			MemFnc.6										:= SingleBlockTrigNext(Execute:= InSingleBlockTrigNext);
		END_IF
	ELSIF NOT SingleBlockTrigNext(Execute:= InSingleBlockTrigNext)
	THEN
		MemDone												:= TRUE;
		MemFnc.6											:= FALSE;
	END_IF
	
	//Reset Intern
	MemFnc.7												:= FALSE;
	
(******************************************************************************)
(* Ctrl Status 																*)
(******************************************************************************)
	Busy													:= CfgBuildExt3DGroup.bBusy
																OR CfgReconfigGroup.bBusy
																OR ItpResetEx2.bBusy
																OR ItpSingleBlock.bBusy
																OR ItpEStopEx.bBusy
																OR ItpStepOnAfterEStopEx.bBusy;
                            						    	
	Done													:= NOT Busy AND MemDone;
                            						    	
	IF done                 	                        	
	THEN                    	                        	
		MemDone												:= FALSE;
	END_IF                  	                        	
                                                        	
	(* Error Output *)                                  	
	IF Busy                                             	
	THEN                                                	
		Error												:= FALSE;
		ErrorId												:= 0;
		ErrorText											:= '';
	ELSIF CfgBuildExt3DGroup.bErr                       	
		AND CfgBuildExt3DGroup.bExecute                 	
	THEN                                                	
		Error												:= TRUE;
		ErrorId												:= CfgBuildExt3DGroup.nErrID;
		ErrorText											:= CONCAT('CfgBuildExt3DGroup ErrorId: ', UDINT_TO_STRING(Errorid));
                                                        	
	ELSIF CfgReconfigGroup.bErr                         	
		AND CfgReconfigGroup.bExecute                   	
	THEN                                                	
		Error												:= TRUE;
		ErrorId												:= CfgReconfigGroup.nErrID;
		ErrorText											:= CONCAT('CfgReconfigGroup ErrorId: ', UDINT_TO_STRING(Errorid));
                                                        	
	ELSIF ItpEStopEx.bErr                               	
		AND ItpEStopEx.bExecute                         	
	THEN                                                	
		Error												:= TRUE;
		ErrorId												:= ItpEStopEx.nErrID;
		ErrorText											:= CONCAT('ItpEStopEx ErrorId: ', UDINT_TO_STRING(Errorid));
                                                        	
	ELSIF ItpStepOnAfterEStopEx.bErr                    	
		AND ItpStepOnAfterEStopEx.bExecute              	
	THEN                                                	
		Error												:= TRUE;
		ErrorId												:= ItpStepOnAfterEStopEx.nErrID;
		ErrorText											:= CONCAT('ItpStepOnAfterEStopEx ErrorId: ', UDINT_TO_STRING(Errorid));
                                                        	
	ELSIF ItpResetEx2.bErr                              	
		AND ItpResetEx2.bExecute                        	
	THEN                                                	
		Error												:= TRUE;
		ErrorId												:= ItpResetEx2.nErrID;
		ErrorText											:= CONCAT('ItpResetEx2 ErrorId: ', UDINT_TO_STRING(Errorid));
                                    	
	ELSIF ItpSingleBlock.bErr                           	
		AND(ItpSingleBlock.bExecuteModeChange OR ItpSingleBlock.bTriggerNext)            	
	THEN                                                	
		Error												:= TRUE;
		ErrorId												:= ItpSingleBlock.nErrID;
		ErrorText											:= CONCAT('ItpSingleBlock ErrorId: ', UDINT_TO_STRING(Errorid));
                                                        	
	ELSIF rNCIRef.NciToPlc.ErrorCode <> 0               	
	THEN                                                	
		Error												:= TRUE;
		ErrorId												:= rNCIRef.NciToPlc.ErrorCode;
		ErrorText											:= CONCAT('NCI Grp ErrorId: ', UDINT_TO_STRING(Errorid));
	ELSE                    						    	
		Error												:= FALSE;
		ErrorId												:= 0;
		ErrorText											:= '';
	END_IF                  	

(********************************************************************************************************)

METHOD PUBLIC reset : BOOL //Return value = TRUE if busy
//required parameter
//rNCIRef
VAR_INPUT
	Execute													:	BOOL;
END_VAR
IF NOT __ISVALIDREF(rNCIRef) 
THEN
	Busy													:= NOT Error;
	ErrorId													:= E_AdsErr.DEVICE_INVALIDPARM;
	Error													:= TRUE;
	Done													:= FALSE;
	ErrorText												:= 'Reference to rNCIRef invalid (0)';
	RETURN;	                							
END_IF

	IF Execute
	THEN
		MemFnc.7											:= TRUE;//Reset intern
		Error												:=FALSE;
		ErrorId												:= 0;
		ItpResetEx2.bExecute 								:= rNCIRef.NciToPlc.ErrorCode <> 0;
	ELSIF NOT ItpSingleBlock.bBusy      					
	THEN                                					
		Error												:=	FALSE;
		ErrorId												:= 0;
		ItpResetEx2.bExecute 								:= FALSE;
	END_IF

	ItpResetEx2(
		bExecute	:= ,
		tTimeOut	:= ,
		sNciToPlc:= rNCIRef.NciToPlc,
		bBusy		=> Busy,
		bErr		=> ,
		nErrId	=> );

	Done													:= NOT ItpResetEx2.bBusy
																AND NOT ItpResetEx2.bErr
																AND ItpResetEx2.bExecute;

	IF NOT Busy
	THEN
		IF ItpResetEx2.bExecute
		THEN
			Error											:=	ItpResetEx2.bErr;
			ErrorId											:= ItpResetEx2.nErrId;
			ErrorText										:= SEL(Error , '' ,  CONCAT('Error ItpResetEx2 id: ',  UDINT_TO_STRING(Errorid)));
		END_IF                          					
		IF NOT Execute                  					
		THEN                            	
			MemFnc.4										:= FALSE ;
			ItpResetEx2(bExecute := FALSE, sNciToPlc:= rNCIRef.NciToPlc);
		END_IF
	END_IF
	
	reset													:= Busy;
END_METHOD

METHOD singleBlockModeChange : BOOL //Return = Busy
VAR_INPUT
	Execute													:	BOOL;
	SingleBlockMode											:	E_ItpSingleBlockMode;
END_VAR
IF NOT __ISVALIDREF(rNCIRef) 
THEN
	Busy													:= NOT Error;
	ErrorId													:= E_adsErr.DEVICE_INVALIDPARM;
	Error													:= TRUE;
	Done													:= FALSE;
	ErrorText												:= 'Reference to rNCIRef invalid (0)';
	RETURN;
END_IF
	
	IF Execute
	THEN
		Error												:=	FALSE;
		ErrorId												:= 0;
		ItpSingleBlock.bExecuteModeChange 					:= TRUE;
	ELSIF NOT ItpSingleBlock.bBusy	    					
	THEN                                					
		Error												:=	FALSE;
		ErrorId												:= 0;
		ItpSingleBlock.bExecuteModeChange 					:= FALSE;

	END_IF
	
	THIS^.SingleBlockMode									:= SingleBlockMode;
									
	ItpSingleBlock(
		bExecuteModeChange	:= ,
		nMode				:= SingleBlockMode,
		bTriggerNext		:=  ,
		tTimeOut			:= ,
		sNciToPlc			:= rNCIRef.NciToPlc,
		bBusy				=> Busy,
		bErr				=> ,
		nErrId				=> );

	Done													:= NOT ItpSingleBlock.bBusy
																AND NOT ItpSingleBlock.bErr
																AND ItpSingleBlock.bExecuteModeChange;

	IF NOT Busy
	THEN
		IF ItpSingleBlock.bExecuteModeChange
		THEN
			Error											:=	ItpSingleBlock.bErr;
			ErrorId											:= ItpSingleBlock.nErrId;
			ErrorText										:= CONCAT('Error ItpSingleBlock id: ',  UDINT_TO_STRING(Errorid));
		END_IF
		IF NOT Execute
		THEN
			MemFnc.5										:= FALSE;
			ItpSingleBlock(bExecuteModeChange := FALSE, sNciToPlc:= rNCIRef.NciToPlc);
		END_IF
	END_IF
	
	SingleBlockModeChange									:= Busy;
END_METHOD

METHOD PUBLIC singleBlockTrigNext : BOOL //Return value = TRUE if busy
//required parameter
//rNCIRef
VAR_INPUT
	Execute													:	BOOL;
END_VAR
IF NOT __ISVALIDREF(rNCIRef) 
THEN
	Busy													:= NOT Error;
	ErrorId													:= E_AdsErr.DEVICE_INVALIDPARM;
	Error													:= TRUE;
	Done													:= FALSE;
	ErrorText												:= 'Reference to rNCIRef invalid (0)';
	RETURN;
END_IF
	
	IF Execute
	THEN
		Error												:=	FALSE;
		ErrorId												:= 0;
		ItpSingleBlock.bTriggerNext 						:= TRUE ;
	ELSIF NOT ItpSingleBlock.bBusy	    					
	THEN                                					
		Error												:=	FALSE;
		ErrorId												:= 0;
		ItpSingleBlock.bTriggerNext 						:= FALSE;

	END_IF

	ItpSingleBlock(
		bExecuteModeChange	:= ,
		nMode				:= SingleBlockMode,
		bTriggerNext		:=  ,
		tTimeOut			:= ,
		sNciToPlc			:= rNCIRef.NciToPlc,
		bBusy				=> Busy,
		bErr				=> ,
		nErrId				=> );

	Done												:= NOT ItpSingleBlock.bBusy
															AND NOT ItpSingleBlock.bErr
															AND ItpSingleBlock.bTriggerNext;

	IF NOT Busy
	THEN
		IF ItpSingleBlock.bTriggerNext
		THEN
			Error										:=	ItpSingleBlock.bErr;
			ErrorId										:= ItpSingleBlock.nErrId;
			ErrorText									:= CONCAT('Error ItpSingleBlock id: ',  UDINT_TO_STRING(Errorid));
		END_IF
		IF NOT Execute
		THEN
			MemFnc.6									:= FALSE;
			ItpSingleBlock(bTriggerNext := FALSE, sNciToPlc:= rNCIRef.NciToPlc);
		END_IF
	END_IF
	
	SingleBlockTrigNext									:= Busy;
END_METHOD

END_FUNCTION_BLOCK

// ---- POUs/Motion/TF5100-NCI/01_Main/NciGrp.TcPOU
{attribute 'no_check'}
//Nci group FB used to build,reconfig Nci groups as well to add and econfig single axis for group
//based on Tc2_NCI
FUNCTION_BLOCK NciGrp EXTENDS FbBase
VAR_OUTPUT CONSTANT
	FNC_BUILD												:	INT := 0; //Build Nci Grp
	FNC_RECONFIG											:	INT := 1; //Reconfig/loose group
	FNC_ADD_AXIS											:	INT := 2; //Add axis to group 
	FNC_RECONFIG_AXIS										:	INT := 3; //Reconfig axis out of grp
END_VAR                     								
VAR_INPUT                   								
	Fnc														:	INT (FNC_BUILD..FNC_RECONFIG_AXIS):= FNC_BUILD;
	XAxisId													: UDINT := 0;
	YAxisId													: UDINT := 0;
	ZAxisId													: UDINT := 0;
	Q1AxisId												: UDINT := 0;
	Q2AxisId												: UDINT := 0;
	Q3AxisId												: UDINT := 0;
	Q4AxisId												: UDINT := 0;
	Q5AxisId												: UDINT := 0;
	AxisIndex												:	NCI_AXCONFIG ;//contains the location of the axis within the group to add or release axis into group 
	rNCIRef													:	REFERENCE TO NCI_REF := 0;
END_VAR                         							
VAR_IN_OUT                      							
END_VAR                         							
VAR_OUTPUT                      							
	ErrorText												:	STRING(40);
END_VAR
VAR
(* Buffer **************************************************************************)
	MemFnc													:	INT := -1;

(* Trigger *)

(* Instanzierung der MC Bausteine *******************************************************)
	CfgBuildExt3DGroup										:	CfgBuildExt3DGroup := (tTimeOut	:= DEFAULT_ADS_TIMEOUT);
	CfgReconfigGroup										:	CfgReconfigGroup := (tTimeOut	:= DEFAULT_ADS_TIMEOUT);
	CfgReconfigAxis											:	CfgReconfigAxis := (tTimeOut	:= DEFAULT_ADS_TIMEOUT);
	CfgAddAxisToGroup										:	CfgAddAxisToGroup:= (tTimeOut	:= DEFAULT_ADS_TIMEOUT);

(* Dummy Speicher **********************************************************)
	K														:	UDINT;
END_VAR

	(* Nci Group control																*)
	(************************************************************************************)

(* Execute ***************************************************************************************)
	rtExecute(CLK := Execute );
	IF rtExecute.Q
		AND MemFnc < 0
	THEN
		MemFnc 												:= Fnc;
		Busy												:= TRUE;
		Done												:= FALSE;
		Error												:= FALSE;
		ErrorID												:= 0;
		ErrorText											:= '';
	END_IF

(* Call Method ***********************************************************************************)
	CASE MemFnc OF
	FNC_BUILD							:	
		Build(Execute	:= Execute);
			
	FNC_RECONFIG						:	
		Reconfig(Execute := Execute);
		
	FNC_ADD_AXIS						:
		CASE AxisIndex OF
		1:	K 												:= XAxisId;
		2:	K 												:= YAxisId;
		3:	K 												:= ZAxisId;
		4:	K 												:= Q1AxisId;
		5:	K 												:= Q2AxisId;
		6:	K 												:= Q3AxisId;
		7:	K 												:= Q4AxisId;
		8:	K 												:= Q5AxisId;
		ELSE
			K 												:= 0;
		END_CASE
		
		AddAxis(
			Execute		:= Execute,
			AxisIndex	:= AxisIndex,
			AxisId		:= k); //location of axis within a group

	FNC_RECONFIG_AXIS					:	

		CASE AxisIndex OF
		1 : K 												:= XAxisId;
		2:	K 												:= YAxisId;
		3:	K 												:= ZAxisId;
		4:	K 												:= Q1AxisId;
		5:	K 												:= Q2AxisId;
		6:	K 												:= Q3AxisId;
		7:	K 												:= Q4AxisId;
		8:	K 												:= Q5AxisId;
		ELSE
			K 												:= 0;
		END_CASE

		ReconfigAxis(
			Execute	:= Execute, 
			AxisId	:= K);
		
	-1:
		IF NOT Execute
		THEN
			Busy											:= FALSE;
			Done											:= FALSE;
			Error											:= FALSE;
			ErrorID											:= 0;
			ErrorText										:= '';
		END_IF                              				
	ELSE                                    				
		Busy												:= FALSE;
		Done												:= FALSE;
		Error												:= Execute;
		ErrorID												:= E_AdsErr.DEVICE_INVALIDPARM;
		ErrorText											:= CONCAT('invalid parameter value(s) Fnc no: ' , INT_TO_STRING(MemFnc));
	END_CASE


(**************************************************************************************************)

METHOD PUBLIC addAxis : BOOL //Return value = TRUE if busy
//required parameter
//rNCIRef
//AxisIndex -> XAxisId..Q5AxisId
VAR_INPUT
	Execute													:	BOOL;
	AxisIndex												:	NCI_AXCONFIG; //contains the location of the axis within the group
	AxisId													:	UDINT; //Axis ID which should be added to group - if 0 then ID of input parameters is used based on parameter AxisIndex
END_VAR
	MemFnc													:= FNC_ADD_AXIS;
	THIS^.Execute											:= Execute;
	THIS^.AxisIndex											:= AxisIndex;
	
IF NOT __ISVALIDREF(rNCIRef) 
THEN
	Busy													:= NOT Error;
	Error													:= TRUE;
	ErrorId													:= E_adsErr.DEVICE_INVALIDPARM;
	Done													:= FALSE;
	ErrorText												:= 'Reference to rNCIRef invalid (0)';
	MemFnc													:= SEL(Execute , -1 ,MemFnc);
	RETURN;
END_IF

	IF Execute
	THEN
		Error												:=	FALSE;
		ErrorId												:= 0;
		CfgAddAxisToGroup.bExecute 							:= TRUE;
	ELSIF NOT CfgAddAxisToGroup.bBusy   					
	THEN                                					
		Error												:=	FALSE;
		ErrorId												:= 0;
		CfgAddAxisToGroup.bExecute 							:= FALSE;

	END_IF
	
	IF AxisId > 0
	THEN
		CfgAddAxisToGroup.nAxisId							:= AxisId;
	ELSE		
		CASE AxisIndex OF
		1:	CfgAddAxisToGroup.nAxisId 						:= XAxisId ;
		2:	CfgAddAxisToGroup.nAxisId 						:= YAxisId ;
		3:	CfgAddAxisToGroup.nAxisId 						:= ZAxisId ;
		4:	CfgAddAxisToGroup.nAxisId 						:= Q1AxisId ;
		5:	CfgAddAxisToGroup.nAxisId 						:= Q2AxisId ;
		6:	CfgAddAxisToGroup.nAxisId 						:= Q3AxisId ;
		7:	CfgAddAxisToGroup.nAxisId 						:= Q4AxisId ;
		8:	CfgAddAxisToGroup.nAxisId 						:= Q5AxisId ;
		ELSE
			CfgAddAxisToGroup.nAxisId 						:= 0;
		END_CASE
	END_IF
	
	CfgAddAxisToGroup(
		bExecute	:= ,
		nGroupId	:= rNCIRef.NciToPlc.GrpId,
		nAxisId		:= ,
		nIndex		:= DINT_TO_UDINT(AxisIndex),
		tTimeOut	:= ,
		bBusy		=> busy,
		bErr		=> ,
		nErrId		=> );

	Done													:= NOT CfgAddAxisToGroup.bBusy
																AND NOT CfgAddAxisToGroup.bErr
																AND CfgAddAxisToGroup.bExecute;
                                        					
	IF NOT Busy                                         	
	THEN                                                	
		IF CfgAddAxisToGroup.bExecute                   	
		THEN                                            	
			Error											:=	CfgAddAxisToGroup.bErr;
			ErrorId											:= CfgAddAxisToGroup.nErrId;
			ErrorText										:= SEL(Error , '' ,  CONCAT('Error CfgAddAxisToGroup id: ',  UDINT_TO_STRING(Errorid)));
		END_IF                                          	
		IF NOT Execute                                  	
		THEN                                            	
			MemFnc											:= -1 ;
			CfgAddAxisToGroup(bExecute := FALSE);       	
		END_IF                                          	
	END_IF                                              	
                                                        	
	AddAxis													:= Busy;
END_METHOD

METHOD PUBLIC build : BOOL //Return value = TRUE if busy
//required parameter
//rNCIRef
//XAxisId
//YAxisId
//ZAxisId
//Q1AxisId
//Q2AxisId
//Q3AxisId
//Q4AxisId
//Q5AxisId
VAR_INPUT
	Execute													:	BOOL;
END_VAR
	MemFnc													:= FNC_BUILD;
	THIS^.Execute											:= Execute;
	
IF NOT __ISVALIDREF(rNCIRef) 
THEN
	Busy													:= NOT Error;
	Error													:= TRUE;
	ErrorId													:= E_AdsErr.DEVICE_INVALIDPARM;
	Done													:= FALSE;
	ErrorText												:= 'Reference to rNCIRef invalid (0)';
	MemFnc													:= SEL(Execute , -1 ,MemFnc);
	RETURN;                                             	
END_IF

	IF Execute
	THEN
		Error												:=	FALSE;
		ErrorId												:= 0;
		CfgBuildExt3DGroup.bExecute 						:= TRUE;
	ELSIF NOT CfgBuildExt3DGroup.bBusy  					
	THEN                                					
		Error												:=	FALSE;
		ErrorId												:= 0;
		CfgBuildExt3DGroup.bExecute 						:= FALSE;
                                        	
	END_IF

	CfgBuildExt3DGroup(
		bExecute	:= ,
		nGroupId	:= rNciRef.NciToPlc.GrpId,
		nXAxisId	:= XAxisId,
		nYAxisId	:= YAxisId,
		nZAxisId	:= ZAxisId,
		nQ1AxisId	:= Q1AxisId,
		nQ2AxisId	:= Q2AxisId,
		nQ3AxisId	:= Q3AxisId,
		nQ4AxisId	:= Q4AxisId,
		nQ5AxisId	:= Q5AxisId,
		tTimeOut	:= ,
		bBusy		=> busy,
		bErr		=> ,
		nErrId	=> );

	Done													:= NOT CfgBuildExt3DGroup.bBusy
																AND NOT CfgBuildExt3DGroup.bErr
																AND CfgBuildExt3DGroup.bExecute;
                                        					
	IF NOT Busy
	THEN
		IF CfgBuildExt3DGroup.bExecute
		THEN
			Error											:=	CfgBuildExt3DGroup.bErr;
			ErrorId											:= CfgBuildExt3DGroup.nErrId;
			ErrorText										:= SEL(Error , '' ,  CONCAT('Error CfgBuildExt3DGroup id: ',  UDINT_TO_STRING(Errorid)));
		END_IF
		IF NOT Execute
		THEN
			MemFnc											:= -1 ;
			CfgBuildExt3DGroup(bExecute := FALSE);
		END_IF
	END_IF

	Build													:= Busy;
END_METHOD

METHOD PUBLIC reconfig : BOOL //Return value = TRUE if busy
//required parameter
//rNCIRef
VAR_INPUT
	Execute													:	BOOL;
END_VAR

	MemFnc													:= FNC_RECONFIG;
	THIS^.Execute											:= Execute;
	
IF NOT __ISVALIDREF(rNCIRef) THEN
	Busy													:= NOT Error;
	Error													:= TRUE;
	ErrorId													:= E_AdsErr.DEVICE_INVALIDPARM;
	Done													:= FALSE;
	ErrorText												:= 'Reference to rNCIRef invalid (0)';
	MemFnc													:= SEL(Execute , -1 ,MemFnc);
	RETURN;
END_IF

	IF Execute
	THEN
		Error												:=	FALSE;
		ErrorId												:= 0;
		CfgReconfigGroup.bExecute 							:= TRUE;
	ELSIF NOT CfgReconfigGroup.bBusy    					
	THEN                                					
		Error												:=	FALSE;
		ErrorId												:= 0;
		CfgReconfigGroup.bExecute 							:= FALSE;

	END_IF

	CfgReconfigGroup(
		bExecute	:= ,
		nGroupId	:= rNCIRef.NciToPlc.GrpId,
		tTimeOut	:= ,
		bBusy		=> busy,
		bErr		=> ,
		nErrId		=> );

	Done													:= NOT CfgReconfigGroup.bBusy
																AND NOT CfgReconfigGroup.bErr
																AND CfgReconfigGroup.bExecute;
                                        					
	IF NOT Busy
	THEN
		IF CfgReconfigGroup.bExecute
		THEN
			Error											:=	CfgReconfigGroup.bErr;
			ErrorId											:= CfgReconfigGroup.nErrId;
			ErrorText										:= SEL(Error , '' ,  CONCAT('Error CfgReconfigGroup id: ',  UDINT_TO_STRING(Errorid)));
		END_IF                      						
		IF NOT Execute              						
		THEN                        						
			MemFnc											:= -1 ;
			CfgReconfigGroup(bExecute := FALSE,);
		END_IF
	END_IF
	
	Reconfig												:= Busy;
END_METHOD

METHOD PUBLIC reconfigAxis : BOOL //Return value = TRUE if busy
//required parameter
//rNCIRef
//AxisId
VAR_INPUT
	Execute													:	BOOL;
	AxisId													:	UDINT; //Axis ID which should be released from group - if 0 then ID of input parameters is used based on parameter AxisIndex
END_VAR
	MemFnc													:= FNC_ADD_AXIS;
	THIS^.Execute											:= Execute;
	
IF NOT __ISVALIDREF(rNCIRef) THEN
	Busy													:= NOT Error;
	Error													:= TRUE;
	ErrorId													:= E_AdsErr.DEVICE_INVALIDPARM;
	Done													:= FALSE;
	ErrorText												:= 'Reference to rNCIRef invalid (0)';
	MemFnc													:= SEL(Execute , -1 ,MemFnc);
	RETURN;
END_IF

	IF Execute
	THEN
		Error												:=	FALSE;
		ErrorId												:= 0;
		CfgReconfigAxis.bExecute 							:= TRUE;
	ELSIF NOT CfgReconfigAxis.bBusy     					
	THEN                                					
		Error												:=	FALSE;
		ErrorId												:= 0;
		CfgReconfigAxis.bExecute 							:= FALSE;

	END_IF

	IF AxisId > 0
	THEN
		CfgReconfigAxis.nAxisId								:= AxisId;
	ELSE
		CASE AxisIndex OF
		1:	CfgReconfigAxis.nAxisId 						:= XAxisId ;
		2:	CfgReconfigAxis.nAxisId 						:= YAxisId ;
		3:	CfgReconfigAxis.nAxisId 						:= ZAxisId ;
		4:	CfgReconfigAxis.nAxisId 						:= Q1AxisId ;
		5:	CfgReconfigAxis.nAxisId 						:= Q2AxisId ;
		6:	CfgReconfigAxis.nAxisId 						:= Q3AxisId ;
		7:	CfgReconfigAxis.nAxisId 						:= Q4AxisId ;
		8:	CfgReconfigAxis.nAxisId 						:= Q5AxisId ;
		ELSE
			CfgReconfigAxis.nAxisId 						:= 0;
		END_CASE
	END_IF

	CfgReconfigAxis(
		bExecute	:= ,
		nAxisId		:= ,
		tTimeOut	:= ,
		bBusy		=> busy,
		bErr		=> ,
		nErrId		=> );

	Done													:= NOT CfgReconfigAxis.bBusy
																AND NOT CfgReconfigAxis.bErr
																AND CfgReconfigAxis.bExecute;
                                        					
	IF NOT Busy
	THEN
		IF CfgReconfigAxis.bExecute
		THEN
			Error											:=	CfgReconfigAxis.bErr;
			ErrorId											:= CfgReconfigAxis.nErrId;
			ErrorText										:= SEL(Error , '' ,  CONCAT('Error CfgReconfigAxis id: ',  UDINT_TO_STRING(Errorid)));
		END_IF
		IF NOT Execute
		THEN
			MemFnc											:= -1 ;
			CfgReconfigAxis(bExecute := FALSE);
		END_IF
	END_IF
	
	ReconfigAxis											:= Busy;
END_METHOD

END_FUNCTION_BLOCK

// ---- POUs/Motion/TF5100-NCI/02_Options/MFunctions/NciMFnc.TcPOU
{attribute 'no_check'}
FUNCTION_BLOCK NciMFnc
VAR_OUTPUT CONSTANT 
	MIN_M_FUNC												:	 UINT := 0;
	MAX_M_FUNC												:	 UINT := 159;
	
//Predefined M Functions
	M2_PRG_END												:	UINT := 2;
	M17_END_SUBROUTINE										:	UINT := 17;
	M30_PRG_END_WITH_ALL_MFUNC								:	UINT := 30; 
END_VAR                 									
VAR_INPUT               									
	ConfirmHsk												:	BOOL := FALSE; (* oder Methode benutzen *)
	FastMFuncReset											:	BOOL := FALSE; (* Signal Start Reser der unter FastMFuncNo angegebenen MFunc Nr. *)
	FastMFuncNo												:	UINT (MIN_M_FUNC..MAX_M_FUNC) := MIN_M_FUNC; (* Nr. der MFunktion die Resetet werden soll *)
	rNCIRef													:	REFERENCE TO NCI_REF := 0;
END_VAR                 									
VAR_OUTPUT              	
	HskReq													:	BOOL;
	HskId													:	UINT; 	
	CntActive												:	INT; //Count number of active M fucntions
	Active													:	BOOL; //Rising trigger M-Function active
	No														:	ARRAY[MIN_M_FUNC..MAX_M_FUNC] OF BOOL; (* Array of M-Functions *)
	rtNo													:	ARRAY[MIN_M_FUNC..MAX_M_FUNC] OF BOOL; (* rising trigger of M-Functions *)
END_VAR                     								
VAR
(* Zwischenspeicher ************************************************************)
	MemFnc													:	INT := -1;

(* Deklaration Trigger **********************************************************)

(* Zeiten ******************************************************************)

(* Bausteine ***************************************************************)
	ItpResetFastMFuncEx										:  ItpResetFastMFuncEx := (tTimeOut	:= DEFAULT_ADS_TIMEOUT);

(* Dummy Speicher **********************************************************)
	i														:	UINT := 0;
	OK														:	BOOL;
END_VAR

	(************************************************************************************)
	(*																					*)
	(*		B E C K H O F F   N E W   A U T O M A T I O N   T E C H N O L O G Y    		*)
	(*																					*)
	(*		Eiserstr.5	D-33415 Verl	Germany	phone:	+49-5246-0	www.Beckhoff.Com	*)
    (*																					*)
    (*		Bausteinbeschreibung	:	Auswerten von M-Funktionen						*)
	(*		TwinCAT-Version			:	2.11.x 											*)
	(*		Version					:	V2.0/ 05/20										*)
 	(*		Autor					:	Daniel Schlingmann								*)
	(*		Lib						:	TcNCI.Lib										*)
	(*																					*)
	(************************************************************************************)

(* evaluate M-function with additional acknowledge *********************************************************************)
	HskReq 													:= rNCIRef.NciToPlc.HskMFuncReq.0;
	HskId 													:= SEL(HskReq, 0, rNCIRef.NciToPlc.HskMFuncNo);

	(* Confirm request *)
	rNCIRef.PlcToNci.MFuncGranted.0 						:= (ConfirmHsk OR rNCIRef.PlcToNci.MFuncGranted.0) AND rNCIRef.NciToPlc.HskMFuncReq.0;

(* set all M-function setzen *)
	CntActive												:= 0;
	Active													:= FALSE;
	
	FOR i := MIN_M_FUNC TO MAX_M_FUNC DO
	 	OK	 												:= ItpIsFastMFunc(UINT_TO_INT(i),rNCIRef.NciToPlc) OR rNCIRef.NciToPlc.HskMFuncNo = i AND rNCIRef.NciToPlc.HskMFuncReq.0;
		rtNo[i]												:= NOT No[i] AND OK;
		No[i]												:= OK;
		IF No[i] 
		THEN 
			CntActive										:= CntActive + 1;		
			Active 											:= TRUE; 
		END_IF
	END_FOR

(* reset fast M-functions, ResetFastMFunc can also be used *)
	IF MemFnc < 0
	THEN
		IF FastMFuncReset
		THEN
			MemFnc 											:= 1;
			ResetFastMFunc(FastMFuncNo:= FastMFuncNo);
		END_IF
	ELSE 
		ResetFastMFunc(FastMFuncNo:= FastMFuncNo);		
	END_IF

(************************************************************************************)

METHOD PUBLIC confirm : BOOL //Return value = TRUE if execution finished
//required parameter
//rNCIRef
VAR_INPUT
END_VAR
IF __ISVALIDREF(rNCIRef)
THEN
	rNCIRef.PlcToNci.MFuncGranted.0 						:= rNCIRef.NciToPlc.HskMFuncReq.0;
	Confirm													:= NOT rNCIRef.NciToPlc.HskMFuncReq.0;
ELSE
	Confirm 												:= TRUE;
END_IF
END_METHOD

METHOD PUBLIC resetFastMFunc : BOOL //Return value = TRUE if busy
//required parameter
//rNCIRef
VAR_INPUT
	FastMFuncNo												:	UINT; (* number of M-function, which has to be resetted *)
END_VAR
IF NOT __ISVALIDREF(rNCIRef)
THEN
	ResetFastMFunc											:= FALSE;
	Return;	
END_IF

	IF ItpIsFastMFunc(UINT_TO_INT(FastMFuncNo),rNCIRef.NciToPlc) 
	THEN
		ItpResetFastMFuncEx.bExecute 						:= TRUE;
		MemFnc.0											:= TRUE;
	ELSIF NOT ItpResetFastMFuncEx.bBusy             		
	THEN                                            		
		ItpResetFastMFuncEx.bExecute 						:= FALSE;
	END_IF
	
	THIS^.FastMFuncNo										:= FastMFuncNo;

	ItpResetFastMFuncEx(
		bExecute	:= ,
		nMFuncNo	:= FastMFuncNo,
		tTimeOut	:= ,
		sNciToPlc	:= rNCIRef.NciToPlc,
		bBusy		=> ,
		bErr		=> ,
		nErrId	=> );
		
	IF NOT ItpResetFastMFuncEx.bBusy
	THEN
		IF ItpResetFastMFuncEx.bExecute
		THEN
			;
		//	Error											:=	ItpResetFastMFuncEx.bErr;
		//	ErrorId											:= ItpResetFastMFuncEx.nErrId;
		END_IF
		IF NOT ItpIsFastMFunc(UINT_TO_INT(FastMFuncNo),rNCIRef.NciToPlc) 
		THEN
			MemFnc											:= -1;
			ItpResetFastMFuncEx(bExecute := FALSE , sNciToPlc:= rNCIRef.NciToPlc);
		END_IF
	END_IF
	
	resetFastMFunc											:= ItpResetFastMFuncEx.bBusy;
END_METHOD

END_FUNCTION_BLOCK

// ---- POUs/Motion/TF5100-NCI/02_Options/RParameter/NCiReadWriteRParam.TcPOU
// To Start read or write, set inpult values and call action read/write. Busy and Done show the status of the operation
FUNCTION_BLOCK NCiReadWriteRParam EXTENDS FbBase
VAR_OUTPUT CONSTANT
	FNC_READ												:	INT := 0;
	FNC_WRITE												:	INT := 1;
END_VAR         											
VAR_INPUT       											
	Fnc														:	INT (FNC_READ..FNC_WRITE) := FNC_READ;
  	pAddr    												: 	PVOID; //Address of parameter destination variable
   	Index   												: 	DINT; //Index to parameter to read
   	Count   												: 	DINT; //
	rNCIRef													:	REFERENCE TO NCI_REF := 0;
END_VAR
VAR_OUTPUT
END_VAR
VAR
(* cache *******************************************************************)
	MemFnc													:	INT := -1;

(* trigger *****************************************************************)

(* function-block instances	************************************************)
	ItpReadRParamsEx										:	ItpReadRParamsEx := (tTimeout := DEFAULT_ADS_TIMEOUT);
	ItpWriteRParamsEx										:	ItpWriteRParamsEx := (tTimeout := DEFAULT_ADS_TIMEOUT);

END_VAR

	(* Read/Write Nci group R parameter													*)
	(************************************************************************************)

(* Execute ******************************************************************************)
	rtExecute(CLK := Execute);
	IF rtExecute.Q
		AND MemFnc < 0
	THEN
		MemFnc 												:= SEL(Fnc = FNC_WRITE, FNC_READ , FNC_WRITE) ;
		Busy												:= TRUE;
		Done												:= FALSE;
		Error												:= FALSE;
		ErrorID												:= 0;
	END_IF

(* Call Method ***************************************************************************)
	CASE MemFnc OF
	FNC_READ:
		Read(Execute );

	FNC_WRITE:
		Write(Execute );

	-1:
		IF NOT Execute
		THEN
			Busy											:= FALSE;
			Done											:= FALSE;
			Error											:= FALSE;
			ErrorID											:= 0;
		END_IF                              				
	ELSE                                    				
		Busy												:= FALSE;
		Done												:= FALSE;
		Error												:= Execute;
		ErrorID												:= E_AdsErr.DEVICE_INVALIDPARM;
	END_CASE

(*************************************************************************************************)

METHOD PUBLIC read : BOOL //Return value = TRUE if busy
//required parameter
//pAddr
//Index
//Count
//rNCIRef
VAR_INPUT 
	Execute													:	BOOL;
END_VAR
	MemFnc 													:= FNC_READ;
	This^.Execute											:= Execute;
IF NOT __ISVALIDREF(rNCIRef) OR pAddr = 0 
THEN
	Busy													:= NOT Error;
	ErrorId													:= E_adsErr.DEVICE_INVALIDPARM;
	Error													:= TRUE;
	Done													:= FALSE;
	MemFnc													:= SEL(Execute , -1 ,MemFnc); 
	RETURN;
END_IF
	
	IF Execute
	THEN
		Error												:=	FALSE;
		ErrorId												:= 0;
		ItpReadRParamsEx.bExecute 							:= TRUE;
	ELSIF NOT ItpReadRParamsEx.bBusy    					
	THEN                                					
		Error												:=	FALSE;
		ErrorId												:= 0;
		ItpReadRParamsEx.bExecute 							:= FALSE;

	END_IF

	ItpReadRParamsEx(
		bExecute	:= ,
		pAddr		:= pAddr,
		nIndex		:= Index,
		nCount		:= Count,
		tTimeOut	:= ,
		sNciToPlc	:= rNCIRef.NciToPlc,
		bBusy		=> Busy,
		bErr		=> ,
		nErrId		=> );

	Done													:= NOT ItpReadRParamsEx.bBusy
																AND NOT ItpReadRParamsEx.bErr
																AND ItpReadRParamsEx.bExecute;
                                                        	
	IF NOT Busy                                         	
	THEN                                                	
		IF ItpReadRParamsEx.bExecute                    	
		THEN                                            	
			Error											:=	ItpReadRParamsEx.bErr;
			ErrorId											:= ItpReadRParamsEx.nErrId;
		END_IF                          					
		IF NOT Execute                  					
		THEN                            	            	
			MemFnc											:= -1;
			ItpReadRParamsEx(bExecute := FALSE , sNciToPlc:= rNCIRef.NciToPlc);
		END_IF
	END_IF
	
	read													:= Busy;
END_METHOD

METHOD PUBLIC write : BOOL //Return value = TRUE if busy
//required parameter
//pAddr
//Index
//Count
//rNCIRef
VAR_INPUT
	Execute													:	BOOL;
END_VAR
	MemFnc 													:= FNC_WRITE;
	THIS^.Execute											:= Execute;

IF NOT __ISVALIDREF(rNCIRef) OR pAddr = 0 
THEN
	Busy													:= NOT Error;
	ErrorId													:= E_adsErr.DEVICE_INVALIDPARM;
	Error													:= TRUE;
	Done													:= FALSE;
	MemFnc													:= SEL(Execute , -1 ,MemFnc); 
	RETURN;
END_IF

	IF Execute
	THEN
		Error												:=	FALSE;
		ErrorId												:= 0;
		ItpWriteRParamsEx.bExecute 							:= TRUE;
	ELSIF NOT ItpWriteRParamsEx.bBusy   					
	THEN                                					
		Error												:=	FALSE;
		ErrorId												:= 0;
		ItpWriteRParamsEx.bExecute 							:= FALSE;

	END_IF

	ItpWriteRParamsEx(
		bExecute	:= ,
		pAddr		:= pAddr,
		nIndex		:= Index,
		nCount		:= Count,
		tTimeOut	:= ,
		sNciToPlc	:= rNCIRef.NciToPlc,
		bBusy		=> Busy,
		bErr		=> ,
		nErrId		=> );

	Done													:= NOT ItpWriteRParamsEx.bBusy
																AND NOT ItpWriteRParamsEx.bErr
																AND ItpWriteRParamsEx.bExecute;
                                        					
	IF NOT Busy
	THEN
		IF ItpWriteRParamsEx.bExecute
		THEN
			Error											:=	ItpWriteRParamsEx.bErr;
			ErrorId											:= ItpWriteRParamsEx.nErrId;
		END_IF                          					
		IF NOT Execute                  					
		THEN                            	
			MemFnc											:= -1;
			ItpWriteRParamsEx(bExecute := FALSE, sNciToPlc:= rNCIRef.NciToPlc);
		END_IF
	END_IF
	
	write													:= Busy;
END_METHOD

END_FUNCTION_BLOCK

// ---- POUs/_Miscellaneous/ERROR_HDL.TcPOU
{attribute 'no_check'}
//Error handle object to collect/provide additional error information like state , function name, id or information text 
FUNCTION_BLOCK ERROR_HDL
VAR_INPUT
	Flag													:	BOOL := FALSE; 	//Error is active
	SourceId												: 	UDINT := 0; 	//Source ID for EventLogger if neede
	EventClass												:	E_TcEventClass := TC2_SYSTEM.TCEVENTCLASS_ALARM;
{attribute 'displaymode':='hex'}
	Id														:	DINT := 0;	//Error id 
	State													:	DINT := 0;	//State where error occures
	Text													:	STRING(MAX_STRING_LENGTH) := '';	//Information text 
	Fnc														:	STRING := '';	//Function name of error source
END_VAR
VAR_OUTPUT
END_VAR
VAR
END_VAR

;

//Reset all entrys to zero/empty
METHOD PUBLIC reset : BOOL  //Return value = TRUE if execution finished
VAR_INPUT
END_VAR
flag 														:= FALSE;
SourceId													:=0;
Eventclass 														:= TC2_SYSTEM.TCEVENTCLASS_NONE;
id															:=0;
state														:=0;
text														:='';
fnc															:='';
Reset														:= TRUE;
END_METHOD

METHOD PUBLIC set : BOOL
VAR_INPUT
	Id														:	DINT := 0;	//Error id 
	State													:	DINT := 0;	//State where error occures
	Text													:	STRING(MAX_STRING_LENGTH) := '';	//Information text 
	Fnc														:	STRING := '';	//Function name of error source
END_VAR
THIS^.Id													:= Id;
THIS^.State													:= State;
THIS^.Text													:= Text;
THIS^.Fnc													:= Fnc;
Flag														:= TRUE;
END_METHOD

END_FUNCTION_BLOCK

// ---- POUs/Motion/TF5100-NCI/02_Options/Error/NciEventHandling.TcPOU
{attribute 'no_check'}
//EventHandlingGrp10 instance used inside
FUNCTION_BLOCK NciEventHandling
VAR CONSTANT
END_VAR                     								
VAR_INPUT                   								
	Enable													:	BOOL := TRUE; (* Show alarm message, warnings or hint. always reported !!! *)
	ConfirmTrig												:	BOOL := FALSE;
	SourceId												:	UDINT := 101200; //TwinCat-NCI channel default multisource Id + Channel id
	ErrorId													:	UDINT := 0;
	Name													:	STRING(30) := '';
	rNci													:	REFERENCE TO NCI_REF := 0;
END_VAR
VAR_OUTPUT
{attribute 'displaymode':='binary'}
	Status													:	DWORD;
	NoOfActiveEvents										:	INT;
END_VAR
VAR
(* Zwischenspeicher ***********************************************)
	QuitInternal 											: BOOL;

(* Timer **********************************************************)

(* Trigger ********************************************************)

(* Bausteine ******************************************************)
	Event													:	EventHandlingGrp10 := (
																	AutoConfirm			:= FALSE, 
																	SetClass 			:= TC2_SYSTEM.TCEVENTCLASS_ALARM );
	ChnEvent												:	NciChnEventHandling;

(* Dummy Speicher *************************************************)
	i														:	INT ;

END_VAR

(* Error message NCI channel to EventLogger 	V1.0	DS	*)
(***********************************************************)

(* Sequence **************************************************************)
IF __ISVALIDREF(rNci) 
THEN
	(* get Quit signal **************************************************)
	IF ConfirmTrig 
	THEN 
		QuitInternal 										:= TRUE; 
	END_IF (* set false see below *)

(* Event Logger Meldungen *****************************************************)
	Event.no[1].Flag 										:= rNci.IsEStopRequested;
	Event.no[2].Flag 										:= rNci.IsFeedFromBackupList;   
	Event.no[3].Flag 										:= rNci.IsMovingBackward;   
	
(*
	Event.no[4].Flag 										:= FALSE;
	Event.no[5].Flag 										:= FALSE;
	Event.no[6].Flag 										:= FALSE;
	Event.no[7].Flag 										:= FALSE;
	Event.no[8].Flag 										:= FALSE;
	Event.no[9].Flag 										:= FALSE;
	Event.no[10].Flag 										:= FALSE;
*)
(* workl Event Ctrl *************************************************)
	IF Event.no[1].Text2 <> Name OR Event.no[1].Text2 <> ''
	THEN
		//Init EventClass
		Event.no[1].eClass 									:= TC2_SYSTEM.TCEVENTCLASS_HINT;
		Event.no[2].eClass 									:= TC2_SYSTEM.TCEVENTCLASS_STATEINFO;
		Event.no[3].eClass 									:= TC2_SYSTEM.TCEVENTCLASS_STATEINFO;

		(* Init Name *)
		FOR i := Event.MIN_EVENT TO Event.MAX_EVENT DO
			Event.no[i].Text2								:= SEL(LEN(name)>1,CONCAT('Channel id:',DWORD_TO_STRING(rNci.NciToPlc.ChnId)),name);
		END_FOR
	END_IF

	Event(
		ConfirmTrig := ConfirmTrig,
		Disable		:= NOT Enable,
		SourceId	:= SourceId + rNci.NciToPlc.ChnId,
		Status	 	=> );	

(* Send ErrorId Message Text **********************************)
	ChnEvent(
		ConfirmTrig	:= NOT Enable OR QuitInternal OR ErrorId = 0 AND ChnEvent.State <> 0,
		Name		:= name,
		ChannelId	:= rNci.NciToPlc.ChnId,
		SourceId	:= Event.SourceId,
		Flag		:= ErrorId > 0 AND Enable,
		ErrorID		:= ErrorId,
		State		=> );

(* EventStatus *************************************************)
	Status													:= ChnEvent.Status OR Event.Status;
	NoOfActiveEvents										:= Event.NoOfActiveEvents + SEL(ChnEvent.Status.31 , 0, 1);

(* Error unkonw pointer or channel id *****************************)
ELSE
	NoOfActiveEvents										:= 0;
	ChnEvent(Flag := FALSE, ConfirmTrig := ChnEvent.State <> 0);
	Event(Disable := TRUE, Status =>  ); 
	Status													:= ChnEvent.Status OR Event.Status;
END_IF

(* Default reset Quit Internal *******************************)
	QuitInternal 											:= FALSE;

(**************************************************************)

METHOD PUBLIC confirm : bool  //Return value = TRUE if execution finished 
VAR_INPUT
END_VAR
QuitInternal 												:= TRUE;
confirm														:= TRUE;
END_METHOD

END_FUNCTION_BLOCK

// ---- POUs/Motion/TF5100-NCI/02_Options/Error/NciChnEventHandling.TcPOU
{attribute 'no_check'}
FUNCTION_BLOCK NciChnEventHandling
VAR_INPUT
	Flag													:	BOOL := FALSE;
	ConfirmTrig												:	BOOL;
	MsgId													:	UDINT := 200; //Default
	SourceId												:	UDINT := 101200;
	ChannelId												:	DWORD := 2;
{attribute 'displaymode':='hex'}
	ErrorId													:	UDINT;
	Name													: 	STRING(20);
END_VAR                         							
VAR_OUTPUT                      							
	State													:	UDINT := TCEVENTSTATE_INVALID;
																		(* TCEVENTSTATE_INVALID  	: WORD := 16#0000; (* Ungültig, kommt auch wenn Event noch nicht gemeldet. *)
																			TCEVENTSTATE_SIGNALED  	: WORD := 16#0001; (* Event ist gemeldet, aber weder gegangen noch quittiert. *)
																			TCEVENTSTATE_RESET  		: WORD := 16#0002; (* Event ist abgemeldet ('gegangen'). *)
																			TCEVENTSTATE_CONFIRMED  : WORD := 16#0010 (16); (* Event ist quittiert. *)
																			TCEVENTSTATE_RESETCON  	: WORD := 16#0012 (17); (* Event ist abgemeldet und quittiert *) *)
{attribute 'displaymode':='binary'}
	Status													:	DWORD; (*	.0 - .8 = event <class id>  / .15 Quit required / .16 = Level 0 , .17 = Level 1 , .18 = Level 2, .......... / .31 active
																			TCEVENTCLASS_NONE			:=0,	(* No class *)
																			TCEVENTCLASS_MAINTENANCE	:=1,	(* Maintenance hint *)
																			TCEVENTCLASS_MESSAGE		:=2,	(* Message *)
																			TCEVENTCLASS_HINT			:=3,	(* Hint *)
																			TCEVENTCLASS_STATEINFO		:=4,	(* State information *)
																			TCEVENTCLASS_INSTRUCTION	:=5,	(* Instruction *)
																			TCEVENTCLASS_WARNING		:=6,	(* Warning *)
																			TCEVENTCLASS_ALARM			:=7,	(* Alarm *)
																			TCEVENTCLASS_PARAMERROR		:=8		(* Parameter error *)  *)
END_VAR
VAR
	AdsEvent												:		ADSLOGEVENT :=(
																		Event			:= FALSE,
																		NETID			:= '',
																		PORT			:= AMSPORT_EVENTLOG,
																		TMOUT 			:= DEFAULT_ADS_TIMEOUT,
																		EventConfigData := (
																					Class 			:= TC2_SYSTEM.TCEVENTCLASS_ALARM,
																					Prio 			:= TCEVENTPRIO_IMPLICIT,
																					ProgId 			:= 'TcEventFormatter.TcXmlFormatter',
																					Flags 			:= 16#0140 (* TCEVENTFLAG_LOG OR TCEVENTFLAG_SRCID *),
																					StreamType 		:= TCEVENTSTREAM_NORMAL (* TCEVENTSTREAM_SIMPLE *),
																					bQuitRequired 	:= FALSE));
                    										
	FormatString 											: STRING(15) := '%s%d%s%s%d%s';
                    										
	pParaArray												: ARRAY [1..6] OF PVOID;
                    										
	Para1													: STRING(30);
	Para2													: UDINT;
	Para3													: STRING(70);
	Para4													: STRING(70);
	Para5													: UDINT;
	Para6													: STRING(20);
	SetClass												: E_TcEventClass := TC2_SYSTEM.TCEVENTCLASS_ALARM;
END_VAR

(* Send axis error text to EventLogger		 							*)
(************************************************************************)

(* Event Config ************************************************)
	IF Status.31 //Message active
	THEN (* work EventLogger *)

		AdsEvent(
			NETID			:= ,(* siehe deklaration *)
			PORT			:= ,(* siehe deklaration *)
			Event			:= NOT AdsEvent.FbCleanup AND(Flag AND Para2 = ErrorID OR AdsEvent.EventState = TCEVENTSTATE_INVALID AND NOT AdsEvent.Quit),
			EventQuit		:= AdsEvent.EventState <> TCEVENTSTATE_INVALID
								AND AdsEvent.EventConfigData.bQuitRequired
								AND NOT AdsEvent.Eventstate.4
								AND NOT AdsEvent.Quit
								AND(
								ConfirmTrig
								OR Para2 <> ErrorID
								OR AdsEvent.EventQuit), (* quit send *)
			EventConfigData	:= ,(* siehe deklaration *)
			EventDataAddress:= ADR(pParaArray),
			EventDataLength	:= ,
			FbCleanup		:= NOT AdsEvent.FbCleanup AND(AdsEvent.Err OR AdsEvent.EventState = TCEVENTSTATE_RESETCON),
			TMOUT			:= ,(* siehe deklaration *)
			EventState		=> ,
			Err				=> ,
			ErrId			=> ,
			Quit			=> );

		IF AdsEvent.Event
			AND AdsEvent.EventState = TCEVENTSTATE_INVALID
		THEN
			State 											:= SEL(Flag, TCEVENTSTATE_RESET, TCEVENTSTATE_SIGNALED);
		ELSIF AdsEvent.Quit
			AND AdsEvent.EventState = TCEVENTSTATE_INVALID
			AND AdsEvent.EventQuit
			OR 
			AdsEvent.FbCleanup		
		THEN
			State 											:= TCEVENTSTATE_RESETCON;
		ELSIF(AdsEvent.Err OR NOT AdsEvent.Event AND AdsEvent.EventState = TCEVENTSTATE_INVALID)
			AND_THEN Gvl.EventHandlingStatistic.CountOut(Status)
		THEN
			State											:= TCEVENTSTATE_INVALID;
		ELSE
			State											:= MAX(State, AdsEvent.EventState);
		END_IF
	
	ELSIF flag AND SourceId > 0
	THEN (* fire event *)
	(*	Type : 2 - Axis Event 201
		%1 User Name 
		%2 	Unique error id (DINT)
		%3	Error text (STRING) ) Bsp.: [S750E20392]
		@V1:%4	Error description (STRING) Bsp.: [S751E20392]
		%5	Logical axis id (DINT)
		@V2:%6	Position OF axis (REAL) or Reserved text 
	
	*)
		Para1 												:= Name;
		Para2 												:= ErrorID;
              												
		Para3 												:= CONCAT('[S','700'); (* SOURCE_TEXT_PTPNCI = 701 *)
		Para3 												:= CONCAT(Para3,'E');
		Para3 												:= CONCAT(Para3,UDINT_TO_STRING(ErrorID));
		Para3 												:= CONCAT(Para3,']');
              												
		Para4 												:= CONCAT('[S','701'); (* SOURCE_DESC_PTPNCI = 701 *)
		Para4 												:= CONCAT(Para4,'E');
		Para4 												:= CONCAT(Para4,UDINT_TO_STRING(ErrorID));
		Para4 												:= CONCAT(Para4,']');
              												
		Para5 												:= ChannelId;
		Para6 												:= ''; (* Reserve *)

		pParaArray[1] 										:= ADR(Para1);
		pParaArray[2] 										:= ADR(Para2);
		pParaArray[3] 										:= ADR(Para3);
		pParaArray[4] 										:= ADR(Para4);
		pParaArray[5] 										:= ADR(Para5);
		pParaArray[6] 										:= ADR(Para6);

		
		AdsEvent.EventConfigData.Id 						:= MsgId; (* MSG_ID = 201 *)
 		AdsEvent.EventConfigData.DataFormatStrAddress 		:= ADR(FormatString);
		AdsEvent.EventConfigData.SourceId 					:= SourceId + ChannelId;
		Status												:= Gvl.EventHandlingStatistic.InitEvent(SetClass , AdsEvent.EventConfigData);	

		IF AdsEvent.Err AND NOT AdsEvent.FbCleanup
		THEN
			AdsEvent(
				Event			:= FALSE,
				EventQuit 		:= FALSE,
				EventDataAddress:= ADR(pParaArray),
				FbCleanup		:= TRUE,
				EventState		=> );
		
		ELSE (* Fire Event *)
			AdsEvent( 	Event			:= FALSE,
						EventQuit 		:= FALSE, 
						FbCleanup 		:= FALSE, 
						EventDataAddress:= ADR(pParaArray));
			AdsEvent( 	Event 	:= TRUE);			
			IF NOT AdsEvent.Err AND_THEN Gvl.EventHandlingStatistic.CountIn(Status) //Add event to statistic and continue if added successfully
			THEN			
				State 										:= TCEVENTSTATE_SIGNALED;
			END_IF
		END_IF
	END_IF

(*****************************************************************)

END_FUNCTION_BLOCK

// ---- POUs/Motion/TF511x-KIN/03_DUTs/Positions/KIN_POSITIONS.TcPOU
{attribute 'no_check'}
FUNCTION_BLOCK KIN_POSITIONS 
VAR_INPUT
	Valid													:	BOOL ;
	MCS														:	KIN_POSITIONS_MCS_DUT; //Values as union
END_VAR
VAR_OUTPUT
END_VAR
VAR
END_VAR

;

METHOD PUBLIC copy : BOOL //Return value = TRUE if execution finished
VAR_IN_OUT
	Source													:	KIN_POSITIONS;
END_VAR
	Valid													:= Source.Valid;
	MCS														:= Source.MCS;
	copy													:= TRUE;
END_METHOD

METHOD PUBLIC delete : BOOL //Return value = TRUE if execution finished - Valid bit will not change
VAR_INPUT
END_VAR
	MCS.A													:= 0.0;
	MCS.B													:= 0.0;
	MCS.C													:= 0.0;
	MCS.X													:= 0.0;
	MCS.Y													:= 0.0;
	MCS.Z													:= 0.0;
	MCS.Q1													:= 0.0;
	MCS.Q2													:= 0.0;
	
	delete													:= TRUE;
END_METHOD

METHOD PUBLIC isInPos : BOOL //Return value = TRUE if axes are within window of checkPos values
VAR_IN_OUT
	CheckPos												:	KIN_POSITIONS_MCS_DUT;
	Window													:	KIN_POSITIONS_MCS_DUT;
END_VAR             										
VAR CONSTANT        										
END_VAR
IsInPos 														:= IsInPosXYZ(CheckPos,Window) AND IsInPosABC(CheckPos,Window);
END_METHOD

METHOD PUBLIC isInPosABC : BOOL //Return value = TRUE if axes are within window of checkPos values
VAR_IN_OUT
	CheckPos												:	KIN_POSITIONS_MCS_DUT;
	Window													:	KIN_POSITIONS_MCS_DUT;
END_VAR                 									
VAR CONSTANT            									
END_VAR
isInPosABC												 	:= CAM(CheckPos.A, MCS.A ,Window.A)
																AND CAM(CheckPos.B, MCS.B ,Window.B)
																AND CAM(CheckPos.C, MCS.C ,Window.C);
END_METHOD

METHOD PUBLIC isInPosByAxisNo : BOOL //Return value = TRUE selected axis is within window of checkPos values
VAR_INPUT
	No					:	INT;
END_VAR
VAR_IN_OUT
	CheckPos			:	KIN_POSITIONS_MCS_DUT;
	Window				:	KIN_POSITIONS_MCS_DUT;
END_VAR
isInPosByAxisNo													:= (CAM(CheckPos.X, MCS.X ,Window.X) OR No <> 1)
																AND (CAM(CheckPos.Y, MCS.Y ,Window.Y) OR No <> 2)
																AND (CAM(CheckPos.Z, MCS.Z ,Window.Z) OR No <> 3)
																AND (CAM(CheckPos.A, MCS.A ,Window.A) OR No <> 4)
																AND (CAM(CheckPos.B, MCS.B ,Window.B) OR No <> 5)
																AND (CAM(CheckPos.C, MCS.C ,Window.C) OR No <> 6)
																AND (CAM(CheckPos.Q1, MCS.Q1 ,Window.Q1) OR No <> 7)
																AND (CAM(CheckPos.Q2, MCS.Q2 ,Window.Q2) OR No <> 8);
END_METHOD

METHOD PUBLIC isInPosExt : BOOL //Return value = TRUE if axes are within window of checkPos values
VAR_INPUT
{attribute 'displaymode':='binary'}
	Config													:	DWORD; //Select value to be checked by bis mask .0=X or A1, .1=Y or A2, .3=Y or A3.....
END_VAR
VAR_IN_OUT
	CheckPos												:	KIN_POSITIONS_MCS_DUT;
	Window													:	KIN_POSITIONS_MCS_DUT;
END_VAR                 									
VAR CONSTANT            									
END_VAR
isInPosExt													:= (CAM(CheckPos.X, MCS.X ,Window.X) OR NOT Config.0)
																AND (CAM(CheckPos.Y, MCS.Y ,Window.Y) OR NOT Config.1)
																AND (CAM(CheckPos.Z, MCS.Z ,Window.Z) OR NOT Config.2)
																AND (CAM(CheckPos.A, MCS.A ,Window.A) OR NOT Config.3)
																AND (CAM(CheckPos.B, MCS.B ,Window.B) OR NOT Config.4)
																AND (CAM(CheckPos.C, MCS.C ,Window.C) OR NOT Config.5)
																AND (CAM(CheckPos.Q1, MCS.Q1 ,Window.Q1) OR NOT Config.6)
																AND (CAM(CheckPos.Q2, MCS.Q2 ,Window.Q2) OR NOT Config.7);
END_METHOD

METHOD PUBLIC isInPosXYZ : BOOL //Return value = TRUE if axes are within window of checkPos values
VAR_IN_OUT
	CheckPos												:	KIN_POSITIONS_MCS_DUT;
	Window													:	KIN_POSITIONS_MCS_DUT;
END_VAR                 									
VAR CONSTANT            									
END_VAR
IsInPosXYZ												 	:= CAM(CheckPos.X, MCS.X ,Window.X)
																AND CAM(CheckPos.Y, MCS.Y ,Window.Y)
																AND CAM(CheckPos.Z, MCS.Z ,Window.Z);
END_METHOD

METHOD PUBLIC reset : BOOL //Delete data and reset valid , TRUE if execution finished
VAR_INPUT
END_VAR
Delete(); 
Valid														:= FALSE;
reset														:= TRUE;
END_METHOD

END_FUNCTION_BLOCK

// ---- POUs/Motion/TF511x-KIN/03_DUTs/Trafo/KIN_CALCTRAFO_AXPOS_PARAM.TcPOU
FUNCTION_BLOCK KIN_CALCTRAFO_AXPOS_PARAM
VAR_INPUT
	In														: 	ARRAY[1..8] OF LREAL;
	Out														: 	ARRAY[1..8] OF LREAL;
	MetaInfoIn												:	U_KinMetaInfo;
	MetaInfoOut												:	U_KinMetaInfo;
END_VAR
VAR_OUTPUT
END_VAR
VAR
END_VAR

METHOD delete : BOOL
VAR_INPUT
END_VAR
MEMSET(ADR(In),0,SIZEOF(In));
MEMSET(ADR(Out),0,SIZEOF(Out));
delete	:= TRUE;
END_METHOD

END_FUNCTION_BLOCK

// ---- POUs/Motion/TF511x-KIN/03_DUTs/Trafo/KIN_STATE_OBSERVER_OID_PARAM.TcPOU
{attribute 'hide'}
FUNCTION_BLOCK KIN_STATE_OBSERVER_OID_PARAM
VAR_INPUT
	oid														:	UDINT := 0; (* Scara State Observer OID *)
	TooltrafoOID											:	UDINT := 0; (* ToolTrafoOID *)
	NextTrafoOID											:	UDINT := 0; (*StaticTrafoOID *)

END_VAR
VAR_OUTPUT

END_VAR
VAR
END_VAR

;

METHOD delete : BOOL
VAR_INPUT
END_VAR
	oid														:= 0;
	TooltrafoOID											:= 0;
	NextTrafoOID											:= 0;
delete	:= TRUE;
END_METHOD

END_FUNCTION_BLOCK

